LIN {X 0,Y 512.253,Z 580.66,A -85,B 0,C 180,E1 4907.429,E2 4907.429} C_VEL
LIN {X 0,Y 512.3,Z 580.66,A -85,B 0,C 180,E1 4912.681,E2 4912.681} C_VEL
LIN {X 0,Y 512.412,Z 580.694,A -85,B 0,C 180,E1 4919.232,E2 4919.232} C_VEL
LIN {X 0,Y 523.878,Z 610.794,A -85,B 0,C 180,E1 4920.286,E2 4920.286} C_VEL
LIN {X 0,Y 523.206,Z 668.635,A -85,B 0,C 180,E1 4921.275,E2 4921.275} C_VEL
LIN {X 0,Y 521.819,Z 705.735,A -85,B 0,C 180,E1 4922.556,E2 4922.556} C_VEL
LIN {X 0,Y 520.117,Z 737.921,A -85,B 0,C 180,E1 4924.318,E2 4924.318} C_VEL
LIN {X 0,Y 518.031,Z 770.325,A -85,B 0,C 180,E1 4926.817,E2 4926.817} C_VEL
LIN {X 0,Y 516.114,Z 799.539,A -85,B 0,C 180,E1 4929.907,E2 4929.907} C_VEL
LIN {X 0,Y 514.641,Z 823.98,A -85,B 0,C 180,E1 4933.388,E2 4933.388} C_VEL
LIN {X 0,Y 513.732,Z 843.903,A -85,B 0,C 180,E1 4937.273,E2 4937.273} C_VEL
LIN {X 0,Y 513.324,Z 857.536,A -85,B 0,C 180,E1 4941.121,E2 4941.121} C_VEL
LIN {X 0,Y 513.093,Z 865.986,A -85,B 0,C 180,E1 4944.937,E2 4944.937} C_VEL
LIN {X 0,Y 513.009,Z 869.513,A -85,B 0,C 180,E1 4948.313,E2 4948.313} C_VEL
LIN {X 0,Y 513.17,Z 869.515,A -85,B 0,C 180,E1 4951.684,E2 4951.684} C_VEL
LIN {X 0,Y 513.084,Z 864.493,A -85,B 0,C 180,E1 4955.907,E2 4955.907} C_VEL
LIN {X 0,Y 513.297,Z 854.958,A -85,B 0,C 180,E1 4959.725,E2 4959.725} C_VEL
LIN {X 0,Y 513.845,Z 840.043,A -85,B 0,C 180,E1 4963.586,E2 4963.586} C_VEL
LIN {X 0,Y 514.932,Z 818.765,A -85,B 0,C 180,E1 4967.453,E2 4967.453} C_VEL
LIN {X 0,Y 516.498,Z 792.754,A -85,B 0,C 180,E1 4970.897,E2 4970.897} C_VEL
LIN {X 0,Y 518.496,Z 762.754,A -85,B 0,C 180,E1 4973.845,E2 4973.845} C_VEL
LIN {X 0,Y 520.653,Z 728.929,A -85,B 0,C 180,E1 4976.245,E2 4976.245} C_VEL
LIN {X 0,Y 522.289,Z 696.341,A -85,B 0,C 180,E1 4977.831,E2 4977.831} C_VEL
LIN {X 0,Y 523.448,Z 660.966,A -85,B 0,C 180,E1 4978.906,E2 4978.906} C_VEL
LIN {X 0,Y 522.927,Z 606.604,A -85,B 0,C 180,E1 4979.824,E2 4979.824} C_VEL
LIN {X 0,Y 512.41,Z 580.66,A -85,B 0,C 180,E1 4980.856,E2 4980.856} C_VEL
LIN {X 0,Y 512.162,Z 580.66,A -85,B 0,C 180,E1 4987.298,E2 4987.298} C_VEL
LIN {X 0,Y 512.152,Z 580.66,A -85,B 0,C 180,E1 4992.657,E2 4992.657} C_VEL
LIN {X 0,Y 512.248,Z 580.66,A -85,B 0,C 180,E1 4997.425,E2 4997.425} C_VEL
LIN {X 0,Y 512.288,Z 580.66,A -85,B 0,C 180,E1 5002.678,E2 5002.678} C_VEL
LIN {X 0,Y 512.29,Z 580.66,A -85,B 0,C 180,E1 5008.666,E2 5008.666} C_VEL
LIN {X 0,Y 512.346,Z 580.66,A -85,B 0,C 180,E1 5013.781,E2 5013.781} C_VEL
LIN {X 0,Y 512.529,Z 580.66,A -85,B 0,C 180,E1 5019.309,E2 5019.309} C_VEL
LIN {X 0,Y 512.44,Z 580.66,A -85,B 0,C 180,E1 5024.63,E2 5024.63} C_VEL
LIN {X 0,Y 512.603,Z 580.66,A -85,B 0,C 180,E1 5029.824,E2 5029.824} C_VEL
LIN {X 0,Y 512.797,Z 580.66,A -85,B 0,C 180,E1 5034.933,E2 5034.933} C_VEL
LIN {X 0,Y 512.816,Z 580.66,A -85,B 0,C 180,E1 5039.997,E2 5039.997} C_VEL
LIN {X 0,Y 512.808,Z 580.66,A -85,B 0,C 180,E1 5045.061,E2 5045.061} C_VEL
LIN {X 0,Y 512.654,Z 580.66,A -85,B 0,C 180,E1 5050.168,E2 5050.168} C_VEL
LIN {X 0,Y 512.572,Z 580.66,A -85,B 0,C 180,E1 5055.36,E2 5055.36} C_VEL
LIN {X 0,Y 512.505,Z 580.66,A -85,B 0,C 180,E1 5060.685,E2 5060.685} C_VEL
LIN {X 0,Y 512.3,Z 580.66,A -85,B 0,C 180,E1 5066.215,E2 5066.215} C_VEL
LIN {X 0,Y 512.314,Z 580.66,A -85,B 0,C 180,E1 5072.011,E2 5072.011} C_VEL
LIN {X 0,Y 512.156,Z 580.66,A -85,B 0,C 180,E1 5078.216,E2 5078.216} C_VEL
LIN {X 0,Y 512.205,Z 580.66,A -85,B 0,C 180,E1 5085.009,E2 5085.009} C_VEL
LIN {X 0,Y 512.33,Z 580.66,A -85,B 0,C 180,E1 5089.967,E2 5089.967} C_VEL
LIN {X 0,Y 512.203,Z 580.66,A -85,B 0,C 180,E1 5095.965,E2 5095.965} C_VEL
LIN {X 0,Y 512.325,Z 580.66,A -85,B 0,C 180,E1 5102.065,E2 5102.065} C_VEL
LIN {X 0,Y 512.487,Z 581.105,A -85,B 0,C 180,E1 5106.168,E2 5106.168} C_VEL
LIN {X 0,Y 520.386,Z 606.411,A -85,B 0,C 180,E1 5107.997,E2 5107.997} C_VEL
LIN {X 0,Y 518.562,Z 636.165,A -85,B 0,C 180,E1 5110.12,E2 5110.12} C_VEL
LIN {X 0,Y 516.609,Z 662.595,A -85,B 0,C 180,E1 5112.838,E2 5112.838} C_VEL
LIN {X 0,Y 514.974,Z 684.992,A -85,B 0,C 180,E1 5116.076,E2 5116.076} C_VEL
LIN {X 0,Y 514.025,Z 701.113,A -85,B 0,C 180,E1 5119.369,E2 5119.369} C_VEL
LIN {X 0,Y 513.36,Z 713.574,A -85,B 0,C 180,E1 5123.249,E2 5123.249} C_VEL
LIN {X 0,Y 513.2,Z 719.653,A -85,B 0,C 180,E1 5126.63,E2 5126.63} C_VEL
LIN {X 0,Y 513.129,Z 721.603,A -85,B 0,C 180,E1 5130.001,E2 5130.001} C_VEL
LIN {X 0,Y 513.261,Z 718.398,A -85,B 0,C 180,E1 5134.216,E2 5134.216} C_VEL
LIN {X 0,Y 513.649,Z 709.866,A -85,B 0,C 180,E1 5138.023,E2 5138.023} C_VEL
LIN {X 0,Y 514.382,Z 695.343,A -85,B 0,C 180,E1 5141.851,E2 5141.851} C_VEL
LIN {X 0,Y 515.675,Z 676.023,A -85,B 0,C 180,E1 5145.27,E2 5145.27} C_VEL
LIN {X 0,Y 517.397,Z 652.213,A -85,B 0,C 180,E1 5148.252,E2 5148.252} C_VEL
LIN {X 0,Y 519.312,Z 624.854,A -85,B 0,C 180,E1 5150.69,E2 5150.69} C_VEL
LIN {X 0,Y 519.753,Z 602.818,A -85,B 0,C 180,E1 5152.175,E2 5152.175} C_VEL
LIN {X 0,Y 512.463,Z 580.66,A -85,B 0,C 180,E1 5153.799,E2 5153.799} C_VEL
LIN {X 0,Y 512.211,Z 580.66,A -85,B 0,C 180,E1 5160.055,E2 5160.055} C_VEL
LIN {X 0,Y 512.277,Z 580.66,A -85,B 0,C 180,E1 5166.095,E2 5166.095} C_VEL
LIN {X 0,Y 512.262,Z 580.66,A -85,B 0,C 180,E1 5170.395,E2 5170.395} C_VEL
LIN {X 0,Y 512.215,Z 580.66,A -85,B 0,C 180,E1 5177.354,E2 5177.354} C_VEL
LIN {X 0,Y 512.267,Z 580.66,A -85,B 0,C 180,E1 5182.686,E2 5182.686} C_VEL
LIN {X 0,Y 512.256,Z 580.66,A -85,B 0,C 180,E1 5188.678,E2 5188.678} C_VEL
LIN {X 0,Y 512.315,Z 580.66,A -85,B 0,C 180,E1 5193.786,E2 5193.786} C_VEL
LIN {X 0,Y 512.532,Z 580.66,A -85,B 0,C 180,E1 5199.316,E2 5199.316} C_VEL
LIN {X 0,Y 512.402,Z 580.66,A -85,B 0,C 180,E1 5204.635,E2 5204.635} C_VEL
LIN {X 0,Y 512.58,Z 580.66,A -85,B 0,C 180,E1 5209.83,E2 5209.83} C_VEL
LIN {X 0,Y 512.817,Z 580.66,A -85,B 0,C 180,E1 5214.939,E2 5214.939} C_VEL
LIN {X 0,Y 512.839,Z 580.66,A -85,B 0,C 180,E1 5220.003,E2 5220.003} C_VEL
LIN {X 0,Y 512.786,Z 580.66,A -85,B 0,C 180,E1 5225.068,E2 5225.068} C_VEL
LIN {X 0,Y 512.686,Z 580.66,A -85,B 0,C 180,E1 5230.174,E2 5230.174} C_VEL
LIN {X 0,Y 512.577,Z 580.66,A -85,B 0,C 180,E1 5235.366,E2 5235.366} C_VEL
LIN {X 0,Y 512.513,Z 580.66,A -85,B 0,C 180,E1 5240.692,E2 5240.692} C_VEL
LIN {X 0,Y 512.325,Z 580.66,A -85,B 0,C 180,E1 5246.22,E2 5246.22} C_VEL
LIN {X 0,Y 512.285,Z 580.66,A -85,B 0,C 180,E1 5252.02,E2 5252.02} C_VEL
LIN {X 0,Y 512.168,Z 580.66,A -85,B 0,C 180,E1 5258.088,E2 5258.088} C_VEL
LIN {X 0,Y 509.69,Z 580.66,A -85,B 0,C 180,E1 5259.518,E2 5259.518} C_VEL
LIN {X 0,Y 504.13,Z 580.66,A -85,B 0,C 180,E1 5261.908,E2 5261.908} C_VEL
LIN {X 0,Y 504.239,Z 580.66,A -85,B 0,C 180,E1 5266.505,E2 5266.505} C_VEL
LIN {X 0,Y 504.372,Z 580.66,A -85,B 0,C 180,E1 5271.077,E2 5271.077} C_VEL
LIN {X 0,Y 504.318,Z 580.66,A -85,B 0,C 180,E1 5276.907,E2 5276.907} C_VEL
LIN {X 0,Y 504.516,Z 580.66,A -85,B 0,C 180,E1 5278.767,E2 5278.767} C_VEL
LIN {X 0,Y 516.691,Z 611.482,A -85,B 0,C 180,E1 5279.931,E2 5279.931} C_VEL
LIN {X 0,Y 516.001,Z 667.111,A -85,B 0,C 180,E1 5280.899,E2 5280.899} C_VEL
LIN {X 0,Y 514.493,Z 704.279,A -85,B 0,C 180,E1 5282.191,E2 5282.191} C_VEL
LIN {X 0,Y 512.569,Z 740.82,A -85,B 0,C 180,E1 5284.163,E2 5284.163} C_VEL
LIN {X 0,Y 510.618,Z 770.896,A -85,B 0,C 180,E1 5286.513,E2 5286.513} C_VEL
LIN {X 0,Y 508.548,Z 799.538,A -85,B 0,C 180,E1 5289.595,E2 5289.595} C_VEL
LIN {X 0,Y 506.924,Z 823.979,A -85,B 0,C 180,E1 5293.127,E2 5293.127} C_VEL
LIN {X 0,Y 505.91,Z 843.903,A -85,B 0,C 180,E1 5297.072,E2 5297.072} C_VEL
LIN {X 0,Y 505.476,Z 856.878,A -85,B 0,C 180,E1 5300.746,E2 5300.746} C_VEL
LIN {X 0,Y 505.195,Z 865.986,A -85,B 0,C 180,E1 5304.858,E2 5304.858} C_VEL
LIN {X 0,Y 505.107,Z 869.513,A -85,B 0,C 180,E1 5308.287,E2 5308.287} C_VEL
LIN {X 0,Y 505.266,Z 869.515,A -85,B 0,C 180,E1 5311.71,E2 5311.71} C_VEL
LIN {X 0,Y 505.202,Z 864.492,A -85,B 0,C 180,E1 5315.999,E2 5315.999} C_VEL
LIN {X 0,Y 505.451,Z 854.946,A -85,B 0,C 180,E1 5319.882,E2 5319.882} C_VEL
LIN {X 0,Y 506.033,Z 840.042,A -85,B 0,C 180,E1 5323.799,E2 5323.799} C_VEL
LIN {X 0,Y 507.212,Z 819.028,A -85,B 0,C 180,E1 5327.686,E2 5327.686} C_VEL
LIN {X 0,Y 508.884,Z 793.85,A -85,B 0,C 180,E1 5331.094,E2 5331.094} C_VEL
LIN {X 0,Y 510.995,Z 764.887,A -85,B 0,C 180,E1 5334.021,E2 5334.021} C_VEL
LIN {X 0,Y 512.854,Z 735.228,A -85,B 0,C 180,E1 5336.187,E2 5336.187} C_VEL
LIN {X 0,Y 514.807,Z 698.308,A -85,B 0,C 180,E1 5338.068,E2 5338.068} C_VEL
LIN {X 0,Y 516.207,Z 660.797,A -85,B 0,C 180,E1 5339.253,E2 5339.253} C_VEL
LIN {X 0,Y 515.751,Z 608.845,A -85,B 0,C 180,E1 5340.157,E2 5340.157} C_VEL
LIN {X 0,Y 504.502,Z 580.66,A -85,B 0,C 180,E1 5341.293,E2 5341.293} C_VEL
LIN {X 0,Y 504.25,Z 580.66,A -85,B 0,C 180,E1 5346.759,E2 5346.759} C_VEL
LIN {X 0,Y 504.17,Z 580.66,A -85,B 0,C 180,E1 5353.498,E2 5353.498} C_VEL
LIN {X 0,Y 504.303,Z 580.66,A -85,B 0,C 180,E1 5358.83,E2 5358.83} C_VEL
LIN {X 0,Y 504.32,Z 580.66,A -85,B 0,C 180,E1 5365.354,E2 5365.354} C_VEL
LIN {X 0,Y 504.371,Z 580.66,A -85,B 0,C 180,E1 5371.399,E2 5371.399} C_VEL
LIN {X 0,Y 504.508,Z 580.66,A -85,B 0,C 180,E1 5377.994,E2 5377.994} C_VEL
LIN {X 0,Y 504.663,Z 580.66,A -85,B 0,C 180,E1 5383.089,E2 5383.089} C_VEL
LIN {X 0,Y 504.679,Z 580.66,A -85,B 0,C 180,E1 5389.663,E2 5389.663} C_VEL
LIN {X 0,Y 504.885,Z 580.66,A -85,B 0,C 180,E1 5394.853,E2 5394.853} C_VEL
LIN {X 0,Y 504.915,Z 580.66,A -85,B 0,C 180,E1 5399.997,E2 5399.997} C_VEL
LIN {X 0,Y 504.892,Z 580.66,A -85,B 0,C 180,E1 5405.141,E2 5405.141} C_VEL
LIN {X 0,Y 504.743,Z 580.66,A -85,B 0,C 180,E1 5410.329,E2 5410.329} C_VEL
LIN {X 0,Y 504.644,Z 580.66,A -85,B 0,C 180,E1 5415.607,E2 5415.607} C_VEL
LIN {X 0,Y 504.55,Z 580.66,A -85,B 0,C 180,E1 5421.027,E2 5421.027} C_VEL
LIN {X 0,Y 504.378,Z 580.66,A -85,B 0,C 180,E1 5426.659,E2 5426.659} C_VEL
LIN {X 0,Y 504.312,Z 580.66,A -85,B 0,C 180,E1 5433.098,E2 5433.098} C_VEL
LIN {X 0,Y 504.228,Z 580.66,A -85,B 0,C 180,E1 5438.929,E2 5438.929} C_VEL
LIN {X 0,Y 504.255,Z 580.66,A -85,B 0,C 180,E1 5445.897,E2 5445.897} C_VEL
LIN {X 0,Y 504.362,Z 580.66,A -85,B 0,C 180,E1 5451.08,E2 5451.08} C_VEL
LIN {X 0,Y 504.252,Z 580.66,A -85,B 0,C 180,E1 5456.906,E2 5456.906} C_VEL
LIN {X 0,Y 504.407,Z 580.66,A -85,B 0,C 180,E1 5463.34,E2 5463.34} C_VEL
LIN {X 0,Y 504.539,Z 581.013,A -85,B 0,C 180,E1 5465.648,E2 5465.648} C_VEL
LIN {X 0,Y 513.395,Z 608.606,A -85,B 0,C 180,E1 5467.666,E2 5467.666} C_VEL
LIN {X 0,Y 511.416,Z 638.199,A -85,B 0,C 180,E1 5469.83,E2 5469.83} C_VEL
LIN {X 0,Y 509.29,Z 664.127,A -85,B 0,C 180,E1 5472.552,E2 5472.552} C_VEL
LIN {X 0,Y 507.558,Z 685.323,A -85,B 0,C 180,E1 5475.657,E2 5475.657} C_VEL
LIN {X 0,Y 506.328,Z 702.896,A -85,B 0,C 180,E1 5479.311,E2 5479.311} C_VEL
LIN {X 0,Y 505.616,Z 714.835,A -85,B 0,C 180,E1 5483.146,E2 5483.146} C_VEL
LIN {X 0,Y 505.418,Z 720.857,A -85,B 0,C 180,E1 5486.578,E2 5486.578} C_VEL
LIN {X 0,Y 505.32,Z 722.79,A -85,B 0,C 180,E1 5490.001,E2 5490.001} C_VEL
LIN {X 0,Y 505.489,Z 719.611,A -85,B 0,C 180,E1 5494.281,E2 5494.281} C_VEL
LIN {X 0,Y 505.914,Z 711.171,A -85,B 0,C 180,E1 5498.146,E2 5498.146} C_VEL
LIN {X 0,Y 506.76,Z 696.769,A -85,B 0,C 180,E1 5502.032,E2 5502.032} C_VEL
LIN {X 0,Y 508.234,Z 677.656,A -85,B 0,C 180,E1 5505.499,E2 5505.499} C_VEL
LIN {X 0,Y 510.182,Z 653.532,A -85,B 0,C 180,E1 5508.583,E2 5508.583} C_VEL
LIN {X 0,Y 512.212,Z 627.084,A -85,B 0,C 180,E1 5510.99,E2 5510.99} C_VEL
LIN {X 0,Y 512.777,Z 605.367,A -85,B 0,C 180,E1 5512.493,E2 5512.493} C_VEL
LIN {X 0,Y 504.501,Z 580.66,A -85,B 0,C 180,E1 5514.355,E2 5514.355} C_VEL
LIN {X 0,Y 504.298,Z 580.66,A -85,B 0,C 180,E1 5520.576,E2 5520.576} C_VEL
LIN {X 0,Y 504.39,Z 580.66,A -85,B 0,C 180,E1 5526.751,E2 5526.751} C_VEL
LIN {X 0,Y 504.21,Z 580.66,A -85,B 0,C 180,E1 5531.576,E2 5531.576} C_VEL
LIN {X 0,Y 504.202,Z 580.66,A -85,B 0,C 180,E1 5536.509,E2 5536.509} C_VEL
LIN {X 0,Y 504.338,Z 580.66,A -85,B 0,C 180,E1 5541.081,E2 5541.081} C_VEL
LIN {X 0,Y 504.248,Z 580.66,A -85,B 0,C 180,E1 5546.919,E2 5546.919} C_VEL
LIN {X 0,Y 504.386,Z 580.66,A -85,B 0,C 180,E1 5553.342,E2 5553.342} C_VEL
LIN {X 0,Y 504.57,Z 580.66,A -85,B 0,C 180,E1 5558.974,E2 5558.974} C_VEL
LIN {X 0,Y 504.499,Z 580.66,A -85,B 0,C 180,E1 5564.388,E2 5564.388} C_VEL
LIN {X 0,Y 504.65,Z 580.66,A -85,B 0,C 180,E1 5570.657,E2 5570.657} C_VEL
LIN {X 0,Y 504.846,Z 580.66,A -85,B 0,C 180,E1 5576.576,E2 5576.576} C_VEL
LIN {X 0,Y 504.793,Z 580.66,A -85,B 0,C 180,E1 5581.716,E2 5581.716} C_VEL
LIN {X 0,Y 504.771,Z 580.66,A -85,B 0,C 180,E1 5586.87,E2 5586.87} C_VEL
LIN {X 0,Y 504.713,Z 580.66,A -85,B 0,C 180,E1 5592.083,E2 5592.083} C_VEL
LIN {X 0,Y 504.628,Z 580.66,A -85,B 0,C 180,E1 5597.401,E2 5597.401} C_VEL
LIN {X 0,Y 504.49,Z 580.66,A -85,B 0,C 180,E1 5602.884,E2 5602.884} C_VEL
LIN {X 0,Y 504.366,Z 580.66,A -85,B 0,C 180,E1 5608.601,E2 5608.601} C_VEL
LIN {X 0,Y 504.309,Z 580.66,A -85,B 0,C 180,E1 5614.647,E2 5614.647} C_VEL
LIN {X 0,Y 504.177,Z 580.66,A -85,B 0,C 180,E1 5621.182,E2 5621.182} C_VEL
LIN {X 0,Y 504.13,Z 580.66,A -85,B 0,C 180,E1 5621.908,E2 5621.908} C_VEL
LIN {X 0,Y 500.222,Z 580.66,A -85,B 0,C 180,E1 5623.857,E2 5623.857} C_VEL
LIN {X 0,Y 496.32,Z 580.66,A -85,B 0,C 180,E1 5625.837,E2 5625.837} C_VEL
LIN {X 0,Y 496.42,Z 580.66,A -85,B 0,C 180,E1 5632.216,E2 5632.216} C_VEL
LIN {X 0,Y 496.608,Z 581.359,A -85,B 0,C 180,E1 5638.366,E2 5638.366} C_VEL
LIN {X 0,Y 509.556,Z 615.391,A -85,B 0,C 180,E1 5639.618,E2 5639.618} C_VEL
LIN {X 0,Y 508.758,Z 666.961,A -85,B 0,C 180,E1 5640.55,E2 5640.55} C_VEL
LIN {X 0,Y 507.091,Z 704.06,A -85,B 0,C 180,E1 5641.87,E2 5641.87} C_VEL
LIN {X 0,Y 505.01,Z 740.835,A -85,B 0,C 180,E1 5643.9,E2 5643.9} C_VEL
LIN {X 0,Y 502.786,Z 774.814,A -85,B 0,C 180,E1 5646.58,E2 5646.58} C_VEL
LIN {X 0,Y 500.904,Z 800.388,A -85,B 0,C 180,E1 5649.381,E2 5649.381} C_VEL
LIN {X 0,Y 499.198,Z 823.978,A -85,B 0,C 180,E1 5652.858,E2 5652.858} C_VEL
LIN {X 0,Y 498.11,Z 843.903,A -85,B 0,C 180,E1 5656.866,E2 5656.866} C_VEL
LIN {X 0,Y 497.509,Z 858.68,A -85,B 0,C 180,E1 5661.276,E2 5661.276} C_VEL
LIN {X 0,Y 497.286,Z 867.19,A -85,B 0,C 180,E1 5665.648,E2 5665.648} C_VEL
LIN {X 0,Y 497.23,Z 870,A -85,B 0,C 180,E1 5669.999,E2 5669.999} C_VEL
LIN {X 0,Y 497.302,Z 867.196,A -85,B 0,C 180,E1 5674.349,E2 5674.349} C_VEL
LIN {X 0,Y 497.476,Z 858.684,A -85,B 0,C 180,E1 5678.721,E2 5678.721} C_VEL
LIN {X 0,Y 497.926,Z 845.658,A -85,B 0,C 180,E1 5682.69,E2 5682.69} C_VEL
LIN {X 0,Y 498.973,Z 826.619,A -85,B 0,C 180,E1 5686.694,E2 5686.694} C_VEL
LIN {X 0,Y 500.71,Z 802.092,A -85,B 0,C 180,E1 5690.402,E2 5690.402} C_VEL
LIN {X 0,Y 502.633,Z 777.24,A -85,B 0,C 180,E1 5693.194,E2 5693.194} C_VEL
LIN {X 0,Y 504.826,Z 744.141,A -85,B 0,C 180,E1 5695.869,E2 5695.869} C_VEL
LIN {X 0,Y 506.887,Z 707.945,A -85,B 0,C 180,E1 5697.958,E2 5697.958} C_VEL
LIN {X 0,Y 508.596,Z 670.167,A -85,B 0,C 180,E1 5699.364,E2 5699.364} C_VEL
LIN {X 0,Y 509.328,Z 625.381,A -85,B 0,C 180,E1 5700.239,E2 5700.239} C_VEL
LIN {X 0,Y 508.58,Z 611.103,A -85,B 0,C 180,E1 5700.501,E2 5700.501} C_VEL
LIN {X 0,Y 496.558,Z 580.66,A -85,B 0,C 180,E1 5701.693,E2 5701.693} C_VEL
LIN {X 0,Y 496.248,Z 580.66,A -85,B 0,C 180,E1 5707.759,E2 5707.759} C_VEL
LIN {X 0,Y 496.301,Z 580.66,A -85,B 0,C 180,E1 5714.367,E2 5714.367} C_VEL
LIN {X 0,Y 496.38,Z 580.66,A -85,B 0,C 180,E1 5720.327,E2 5720.327} C_VEL
LIN {X 0,Y 496.377,Z 580.66,A -85,B 0,C 180,E1 5726.824,E2 5726.824} C_VEL
LIN {X 0,Y 496.458,Z 580.66,A -85,B 0,C 180,E1 5732.874,E2 5732.874} C_VEL
LIN {X 0,Y 496.637,Z 580.66,A -85,B 0,C 180,E1 5738.615,E2 5738.615} C_VEL
LIN {X 0,Y 496.647,Z 580.66,A -85,B 0,C 180,E1 5744.128,E2 5744.128} C_VEL
LIN {X 0,Y 496.75,Z 580.66,A -85,B 0,C 180,E1 5749.496,E2 5749.496} C_VEL
LIN {X 0,Y 496.987,Z 580.66,A -85,B 0,C 180,E1 5754.771,E2 5754.771} C_VEL
LIN {X 0,Y 497.022,Z 580.66,A -85,B 0,C 180,E1 5759.997,E2 5759.997} C_VEL
LIN {X 0,Y 496.987,Z 580.66,A -85,B 0,C 180,E1 5765.222,E2 5765.222} C_VEL
LIN {X 0,Y 496.817,Z 580.66,A -85,B 0,C 180,E1 5770.496,E2 5770.496} C_VEL
LIN {X 0,Y 496.733,Z 580.66,A -85,B 0,C 180,E1 5775.862,E2 5775.862} C_VEL
LIN {X 0,Y 496.621,Z 580.66,A -85,B 0,C 180,E1 5781.379,E2 5781.379} C_VEL
LIN {X 0,Y 496.418,Z 580.66,A -85,B 0,C 180,E1 5787.121,E2 5787.121} C_VEL
LIN {X 0,Y 496.405,Z 580.66,A -85,B 0,C 180,E1 5793.166,E2 5793.166} C_VEL
LIN {X 0,Y 496.222,Z 580.66,A -85,B 0,C 180,E1 5799.679,E2 5799.679} C_VEL
LIN {X 0,Y 496.334,Z 580.66,A -85,B 0,C 180,E1 5805.637,E2 5805.637} C_VEL
LIN {X 0,Y 496.403,Z 580.66,A -85,B 0,C 180,E1 5812.208,E2 5812.208} C_VEL
LIN {X 0,Y 496.316,Z 580.66,A -85,B 0,C 180,E1 5818.34,E2 5818.34} C_VEL
LIN {X 0,Y 496.522,Z 580.66,A -85,B 0,C 180,E1 5824.822,E2 5824.822} C_VEL
LIN {X 0,Y 496.596,Z 581.594,A -85,B 0,C 180,E1 5825.148,E2 5825.148} C_VEL
LIN {X 0,Y 506.22,Z 610.107,A -85,B 0,C 180,E1 5827.287,E2 5827.287} C_VEL
LIN {X 0,Y 504.243,Z 640.16,A -85,B 0,C 180,E1 5829.53,E2 5829.53} C_VEL
LIN {X 0,Y 501.927,Z 666.279,A -85,B 0,C 180,E1 5832.334,E2 5832.334} C_VEL
LIN {X 0,Y 500.02,Z 687.497,A -85,B 0,C 180,E1 5835.55,E2 5835.55} C_VEL
LIN {X 0,Y 498.684,Z 704.107,A -85,B 0,C 180,E1 5839.101,E2 5839.101} C_VEL
LIN {X 0,Y 497.871,Z 716.1,A -85,B 0,C 180,E1 5843.038,E2 5843.038} C_VEL
LIN {X 0,Y 497.63,Z 722.064,A -85,B 0,C 180,E1 5846.525,E2 5846.525} C_VEL
LIN {X 0,Y 497.532,Z 723.973,A -85,B 0,C 180,E1 5850.001,E2 5850.001} C_VEL
LIN {X 0,Y 497.714,Z 720.826,A -85,B 0,C 180,E1 5854.348,E2 5854.348} C_VEL
LIN {X 0,Y 498.182,Z 712.466,A -85,B 0,C 180,E1 5858.273,E2 5858.273} C_VEL
LIN {X 0,Y 499.167,Z 698.228,A -85,B 0,C 180,E1 5862.218,E2 5862.218} C_VEL
LIN {X 0,Y 500.797,Z 679.309,A -85,B 0,C 180,E1 5865.736,E2 5865.736} C_VEL
LIN {X 0,Y 502.922,Z 655.399,A -85,B 0,C 180,E1 5868.862,E2 5868.862} C_VEL
LIN {X 0,Y 505.197,Z 627.918,A -85,B 0,C 180,E1 5871.394,E2 5871.394} C_VEL
LIN {X 0,Y 505.961,Z 608.702,A -85,B 0,C 180,E1 5872.729,E2 5872.729} C_VEL
LIN {X 0,Y 496.531,Z 580.66,A -85,B 0,C 180,E1 5874.825,E2 5874.825} C_VEL
LIN {X 0,Y 496.325,Z 580.66,A -85,B 0,C 180,E1 5881.122,E2 5881.122} C_VEL
LIN {X 0,Y 496.4,Z 580.66,A -85,B 0,C 180,E1 5887.443,E2 5887.443} C_VEL
LIN {X 0,Y 496.249,Z 580.66,A -85,B 0,C 180,E1 5893.141,E2 5893.141} C_VEL
LIN {X 0,Y 496.319,Z 580.66,A -85,B 0,C 180,E1 5899.471,E2 5899.471} C_VEL
LIN {X 0,Y 496.378,Z 580.66,A -85,B 0,C 180,E1 5905.163,E2 5905.163} C_VEL
LIN {X 0,Y 496.384,Z 580.66,A -85,B 0,C 180,E1 5911.833,E2 5911.833} C_VEL
LIN {X 0,Y 496.513,Z 580.66,A -85,B 0,C 180,E1 5916.734,E2 5916.734} C_VEL
LIN {X 0,Y 496.728,Z 580.66,A -85,B 0,C 180,E1 5922.32,E2 5922.32} C_VEL
LIN {X 0,Y 496.729,Z 580.66,A -85,B 0,C 180,E1 5929.502,E2 5929.502} C_VEL
LIN {X 0,Y 497.007,Z 580.66,A -85,B 0,C 180,E1 5934.778,E2 5934.778} C_VEL
LIN {X 0,Y 497.044,Z 580.66,A -85,B 0,C 180,E1 5940.003,E2 5940.003} C_VEL
LIN {X 0,Y 496.972,Z 580.66,A -85,B 0,C 180,E1 5945.229,E2 5945.229} C_VEL
LIN {X 0,Y 496.85,Z 580.66,A -85,B 0,C 180,E1 5950.502,E2 5950.502} C_VEL
LIN {X 0,Y 496.725,Z 580.66,A -85,B 0,C 180,E1 5955.869,E2 5955.869} C_VEL
LIN {X 0,Y 496.636,Z 580.66,A -85,B 0,C 180,E1 5961.385,E2 5961.385} C_VEL
LIN {X 0,Y 496.45,Z 580.66,A -85,B 0,C 180,E1 5967.126,E2 5967.126} C_VEL
LIN {X 0,Y 496.388,Z 580.66,A -85,B 0,C 180,E1 5973.175,E2 5973.175} C_VEL
LIN {X 0,Y 496.23,Z 580.66,A -85,B 0,C 180,E1 5979.687,E2 5979.687} C_VEL
LIN {X 0,Y 496.32,Z 580.66,A -85,B 0,C 180,E1 5985.837,E2 5985.837} C_VEL
LIN {X 0,Y 492.364,Z 580.66,A -85,B 0,C 180,E1 5987.811,E2 5987.811} C_VEL
LIN {X 0,Y 488.442,Z 580.66,A -85,B 0,C 180,E1 5989.816,E2 5989.816} C_VEL
LIN {X 0,Y 488.477,Z 580.66,A -85,B 0,C 180,E1 5996.217,E2 5996.217} C_VEL
LIN {X 0,Y 488.598,Z 581.283,A -85,B 0,C 180,E1 5997.887,E2 5997.887} C_VEL
LIN {X 0,Y 502.356,Z 615.662,A -85,B 0,C 180,E1 5999.241,E2 5999.241} C_VEL
LIN {X 0,Y 501.523,Z 666.523,A -85,B 0,C 180,E1 6000.185,E2 6000.185} C_VEL
LIN {X 0,Y 499.741,Z 702.563,A -85,B 0,C 180,E1 6001.48,E2 6001.48} C_VEL
LIN {X 0,Y 497.538,Z 739.366,A -85,B 0,C 180,E1 6003.532,E2 6003.532} C_VEL
LIN {X 0,Y 495.241,Z 772.505,A -85,B 0,C 180,E1 6006.162,E2 6006.162} C_VEL
LIN {X 0,Y 493.21,Z 800.895,A -85,B 0,C 180,E1 6009.188,E2 6009.188} C_VEL
LIN {X 0,Y 491.656,Z 821.333,A -85,B 0,C 180,E1 6012.126,E2 6012.126} C_VEL
LIN {X 0,Y 490.443,Z 840.028,A -85,B 0,C 180,E1 6015.75,E2 6015.75} C_VEL
LIN {X 0,Y 489.744,Z 855.451,A -85,B 0,C 180,E1 6019.967,E2 6019.967} C_VEL
LIN {X 0,Y 489.497,Z 864.486,A -85,B 0,C 180,E1 6023.805,E2 6023.805} C_VEL
LIN {X 0,Y 489.325,Z 869.512,A -85,B 0,C 180,E1 6028.231,E2 6028.231} C_VEL
LIN {X 0,Y 489.474,Z 869.514,A -85,B 0,C 180,E1 6031.765,E2 6031.765} C_VEL
LIN {X 0,Y 489.447,Z 864.492,A -85,B 0,C 180,E1 6036.193,E2 6036.193} C_VEL
LIN {X 0,Y 489.697,Z 855.533,A -85,B 0,C 180,E1 6040.005,E2 6040.005} C_VEL
LIN {X 0,Y 490.467,Z 840.041,A -85,B 0,C 180,E1 6044.246,E2 6044.246} C_VEL
LIN {X 0,Y 491.899,Z 819.149,A -85,B 0,C 180,E1 6048.236,E2 6048.236} C_VEL
LIN {X 0,Y 493.488,Z 796.447,A -85,B 0,C 180,E1 6051.355,E2 6051.355} C_VEL
LIN {X 0,Y 495.696,Z 765.715,A -85,B 0,C 180,E1 6054.444,E2 6054.444} C_VEL
LIN {X 0,Y 497.951,Z 732.522,A -85,B 0,C 180,E1 6056.907,E2 6056.907} C_VEL
LIN {X 0,Y 500.161,Z 696.283,A -85,B 0,C 180,E1 6058.798,E2 6058.798} C_VEL
LIN {X 0,Y 501.796,Z 658.508,A -85,B 0,C 180,E1 6060.018,E2 6060.018} C_VEL
LIN {X 0,Y 501.448,Z 613.288,A -85,B 0,C 180,E1 6060.857,E2 6060.857} C_VEL
LIN {X 0,Y 488.586,Z 580.66,A -85,B 0,C 180,E1 6062.218,E2 6062.218} C_VEL
LIN {X 0,Y 488.323,Z 580.66,A -85,B 0,C 180,E1 6068.168,E2 6068.168} C_VEL
LIN {X 0,Y 488.392,Z 580.66,A -85,B 0,C 180,E1 6074.714,E2 6074.714} C_VEL
LIN {X 0,Y 488.455,Z 580.66,A -85,B 0,C 180,E1 6080.558,E2 6080.558} C_VEL
LIN {X 0,Y 488.464,Z 580.66,A -85,B 0,C 180,E1 6086.515,E2 6086.515} C_VEL
LIN {X 0,Y 488.532,Z 580.66,A -85,B 0,C 180,E1 6092.397,E2 6092.397} C_VEL
LIN {X 0,Y 488.67,Z 580.66,A -85,B 0,C 180,E1 6098.249,E2 6098.249} C_VEL
LIN {X 0,Y 488.73,Z 580.66,A -85,B 0,C 180,E1 6103.864,E2 6103.864} C_VEL
LIN {X 0,Y 488.828,Z 580.66,A -85,B 0,C 180,E1 6109.324,E2 6109.324} C_VEL
LIN {X 0,Y 489.074,Z 580.66,A -85,B 0,C 180,E1 6114.686,E2 6114.686} C_VEL
LIN {X 0,Y 489.122,Z 580.66,A -85,B 0,C 180,E1 6119.997,E2 6119.997} C_VEL
LIN {X 0,Y 489.071,Z 580.66,A -85,B 0,C 180,E1 6125.307,E2 6125.307} C_VEL
LIN {X 0,Y 488.891,Z 580.66,A -85,B 0,C 180,E1 6130.668,E2 6130.668} C_VEL
LIN {X 0,Y 488.761,Z 580.66,A -85,B 0,C 180,E1 6136.861,E2 6136.861} C_VEL
LIN {X 0,Y 488.65,Z 580.66,A -85,B 0,C 180,E1 6142.127,E2 6142.127} C_VEL
LIN {X 0,Y 488.497,Z 580.66,A -85,B 0,C 180,E1 6147.598,E2 6147.598} C_VEL
LIN {X 0,Y 488.454,Z 580.66,A -85,B 0,C 180,E1 6153.778,E2 6153.778} C_VEL
LIN {X 0,Y 488.317,Z 580.66,A -85,B 0,C 180,E1 6160.453,E2 6160.453} C_VEL
LIN {X 0,Y 488.418,Z 580.66,A -85,B 0,C 180,E1 6167.185,E2 6167.185} C_VEL
LIN {X 0,Y 488.436,Z 580.66,A -85,B 0,C 180,E1 6173.43,E2 6173.43} C_VEL
LIN {X 0,Y 488.409,Z 580.66,A -85,B 0,C 180,E1 6179.878,E2 6179.878} C_VEL
LIN {X 0,Y 488.616,Z 581.156,A -85,B 0,C 180,E1 6184.59,E2 6184.59} C_VEL
LIN {X 0,Y 499.064,Z 611.96,A -85,B 0,C 180,E1 6186.938,E2 6186.938} C_VEL
LIN {X 0,Y 497.031,Z 641.874,A -85,B 0,C 180,E1 6189.219,E2 6189.219} C_VEL
LIN {X 0,Y 494.631,Z 667.725,A -85,B 0,C 180,E1 6192.034,E2 6192.034} C_VEL
LIN {X 0,Y 492.518,Z 689.061,A -85,B 0,C 180,E1 6195.325,E2 6195.325} C_VEL
LIN {X 0,Y 491.036,Z 705.495,A -85,B 0,C 180,E1 6198.929,E2 6198.929} C_VEL
LIN {X 0,Y 490.132,Z 717.374,A -85,B 0,C 180,E1 6202.928,E2 6202.928} C_VEL
LIN {X 0,Y 489.849,Z 723.27,A -85,B 0,C 180,E1 6206.469,E2 6206.469} C_VEL
LIN {X 0,Y 489.723,Z 725.16,A -85,B 0,C 180,E1 6210.001,E2 6210.001} C_VEL
LIN {X 0,Y 489.933,Z 722.044,A -85,B 0,C 180,E1 6214.417,E2 6214.417} C_VEL
LIN {X 0,Y 490.459,Z 713.789,A -85,B 0,C 180,E1 6218.405,E2 6218.405} C_VEL
LIN {X 0,Y 491.579,Z 699.686,A -85,B 0,C 180,E1 6222.409,E2 6222.409} C_VEL
LIN {X 0,Y 493.349,Z 680.929,A -85,B 0,C 180,E1 6225.979,E2 6225.979} C_VEL
LIN {X 0,Y 495.56,Z 657.962,A -85,B 0,C 180,E1 6229.05,E2 6229.05} C_VEL
LIN {X 0,Y 497.943,Z 630.97,A -85,B 0,C 180,E1 6231.622,E2 6231.622} C_VEL
LIN {X 0,Y 498.684,Z 610.457,A -85,B 0,C 180,E1 6233.093,E2 6233.093} C_VEL
LIN {X 0,Y 488.61,Z 580.66,A -85,B 0,C 180,E1 6235.34,E2 6235.34} C_VEL
LIN {X 0,Y 488.397,Z 580.66,A -85,B 0,C 180,E1 6241.685,E2 6241.685} C_VEL
LIN {X 0,Y 488.476,Z 580.66,A -85,B 0,C 180,E1 6248.158,E2 6248.158} C_VEL
LIN {X 0,Y 488.372,Z 580.66,A -85,B 0,C 180,E1 6254.721,E2 6254.721} C_VEL
LIN {X 0,Y 488.434,Z 580.66,A -85,B 0,C 180,E1 6260.565,E2 6260.565} C_VEL
LIN {X 0,Y 488.417,Z 580.66,A -85,B 0,C 180,E1 6266.529,E2 6266.529} C_VEL
LIN {X 0,Y 488.48,Z 580.66,A -85,B 0,C 180,E1 6272.401,E2 6272.401} C_VEL
LIN {X 0,Y 488.67,Z 580.66,A -85,B 0,C 180,E1 6278.256,E2 6278.256} C_VEL
LIN {X 0,Y 488.706,Z 580.66,A -85,B 0,C 180,E1 6283.87,E2 6283.87} C_VEL
LIN {X 0,Y 488.808,Z 580.66,A -85,B 0,C 180,E1 6289.33,E2 6289.33} C_VEL
LIN {X 0,Y 489.093,Z 580.66,A -85,B 0,C 180,E1 6294.693,E2 6294.693} C_VEL
LIN {X 0,Y 489.143,Z 580.66,A -85,B 0,C 180,E1 6300.003,E2 6300.003} C_VEL
LIN {X 0,Y 489.056,Z 580.66,A -85,B 0,C 180,E1 6305.314,E2 6305.314} C_VEL
LIN {X 0,Y 488.924,Z 580.66,A -85,B 0,C 180,E1 6310.674,E2 6310.674} C_VEL
LIN {X 0,Y 488.745,Z 580.66,A -85,B 0,C 180,E1 6316.844,E2 6316.844} C_VEL
LIN {X 0,Y 488.659,Z 580.66,A -85,B 0,C 180,E1 6322.122,E2 6322.122} C_VEL
LIN {X 0,Y 488.526,Z 580.66,A -85,B 0,C 180,E1 6327.603,E2 6327.603} C_VEL
LIN {X 0,Y 488.458,Z 580.66,A -85,B 0,C 180,E1 6333.785,E2 6333.785} C_VEL
LIN {X 0,Y 488.332,Z 580.66,A -85,B 0,C 180,E1 6340.46,E2 6340.46} C_VEL
LIN {X 0,Y 488.36,Z 580.66,A -85,B 0,C 180,E1 6345.831,E2 6345.831} C_VEL
LIN {X 0,Y 488.442,Z 580.66,A -85,B 0,C 180,E1 6349.816,E2 6349.816} C_VEL
LIN {X 0,Y 485.942,Z 580.66,A -85,B 0,C 180,E1 6351.328,E2 6351.328} C_VEL
LIN {X 0,Y 480.518,Z 580.66,A -85,B 0,C 180,E1 6353.859,E2 6353.859} C_VEL
LIN {X 0,Y 480.662,Z 581.316,A -85,B 0,C 180,E1 6357.39,E2 6357.39} C_VEL
LIN {X 0,Y 495.167,Z 617.768,A -85,B 0,C 180,E1 6358.884,E2 6358.884} C_VEL
LIN {X 0,Y 494.292,Z 665.78,A -85,B 0,C 180,E1 6359.807,E2 6359.807} C_VEL
LIN {X 0,Y 492.421,Z 701.316,A -85,B 0,C 180,E1 6361.102,E2 6361.102} C_VEL
LIN {X 0,Y 490.059,Z 738.353,A -85,B 0,C 180,E1 6363.184,E2 6363.184} C_VEL
LIN {X 0,Y 487.525,Z 772.575,A -85,B 0,C 180,E1 6365.957,E2 6365.957} C_VEL
LIN {X 0,Y 485.273,Z 802.452,A -85,B 0,C 180,E1 6369.248,E2 6369.248} C_VEL
LIN {X 0,Y 483.489,Z 827.744,A -85,B 0,C 180,E1 6373.023,E2 6373.023} C_VEL
LIN {X 0,Y 482.431,Z 844.396,A -85,B 0,C 180,E1 6376.56,E2 6376.56} C_VEL
LIN {X 0,Y 481.769,Z 858.68,A -85,B 0,C 180,E1 6380.989,E2 6380.989} C_VEL
LIN {X 0,Y 481.517,Z 867.189,A -85,B 0,C 180,E1 6385.505,E2 6385.505} C_VEL
LIN {X 0,Y 481.437,Z 870,A -85,B 0,C 180,E1 6389.998,E2 6389.998} C_VEL
LIN {X 0,Y 481.524,Z 867.195,A -85,B 0,C 180,E1 6394.492,E2 6394.492} C_VEL
LIN {X 0,Y 481.726,Z 858.684,A -85,B 0,C 180,E1 6399.009,E2 6399.009} C_VEL
LIN {X 0,Y 482.34,Z 844.375,A -85,B 0,C 180,E1 6403.448,E2 6403.448} C_VEL
LIN {X 0,Y 483.51,Z 826.502,A -85,B 0,C 180,E1 6407.202,E2 6407.202} C_VEL
LIN {X 0,Y 485.284,Z 801.367,A -85,B 0,C 180,E1 6410.887,E2 6410.887} C_VEL
LIN {X 0,Y 487.529,Z 772.563,A -85,B 0,C 180,E1 6414.043,E2 6414.043} C_VEL
LIN {X 0,Y 489.946,Z 739.612,A -85,B 0,C 180,E1 6416.728,E2 6416.728} C_VEL
LIN {X 0,Y 492.38,Z 702.522,A -85,B 0,C 180,E1 6418.843,E2 6418.843} C_VEL
LIN {X 0,Y 494.315,Z 665.33,A -85,B 0,C 180,E1 6420.207,E2 6420.207} C_VEL
LIN {X 0,Y 494.475,Z 616.025,A -85,B 0,C 180,E1 6421.195,E2 6421.195} C_VEL
LIN {X 0,Y 480.642,Z 580.66,A -85,B 0,C 180,E1 6422.652,E2 6422.652} C_VEL
LIN {X 0,Y 480.395,Z 580.66,A -85,B 0,C 180,E1 6428.915,E2 6428.915} C_VEL
LIN {X 0,Y 480.402,Z 580.66,A -85,B 0,C 180,E1 6433.743,E2 6433.743} C_VEL
LIN {X 0,Y 480.505,Z 580.66,A -85,B 0,C 180,E1 6438.906,E2 6438.906} C_VEL
LIN {X 0,Y 480.491,Z 580.66,A -85,B 0,C 180,E1 6444.733,E2 6444.733} C_VEL
LIN {X 0,Y 480.542,Z 580.66,A -85,B 0,C 180,E1 6449.838,E2 6449.838} C_VEL
LIN {X 0,Y 480.652,Z 580.66,A -85,B 0,C 180,E1 6455.911,E2 6455.911} C_VEL
LIN {X 0,Y 480.867,Z 580.66,A -85,B 0,C 180,E1 6461.709,E2 6461.709} C_VEL
LIN {X 0,Y 480.799,Z 580.66,A -85,B 0,C 180,E1 6467.307,E2 6467.307} C_VEL
LIN {X 0,Y 481.107,Z 580.66,A -85,B 0,C 180,E1 6472.79,E2 6472.79} C_VEL
LIN {X 0,Y 481.379,Z 580.66,A -85,B 0,C 180,E1 6478.2,E2 6478.2} C_VEL
LIN {X 0,Y 481.324,Z 580.66,A -85,B 0,C 180,E1 6483.591,E2 6483.591} C_VEL
LIN {X 0,Y 481.05,Z 580.66,A -85,B 0,C 180,E1 6489.02,E2 6489.02} C_VEL
LIN {X 0,Y 480.94,Z 580.66,A -85,B 0,C 180,E1 6494.532,E2 6494.532} C_VEL
LIN {X 0,Y 480.797,Z 580.66,A -85,B 0,C 180,E1 6500.191,E2 6500.191} C_VEL
LIN {X 0,Y 480.617,Z 580.66,A -85,B 0,C 180,E1 6506.069,E2 6506.069} C_VEL
LIN {X 0,Y 480.557,Z 580.66,A -85,B 0,C 180,E1 6512.256,E2 6512.256} C_VEL
LIN {X 0,Y 480.389,Z 580.66,A -85,B 0,C 180,E1 6518.912,E2 6518.912} C_VEL
LIN {X 0,Y 480.391,Z 580.66,A -85,B 0,C 180,E1 6523.746,E2 6523.746} C_VEL
LIN {X 0,Y 480.497,Z 580.66,A -85,B 0,C 180,E1 6528.902,E2 6528.902} C_VEL
LIN {X 0,Y 480.481,Z 580.66,A -85,B 0,C 180,E1 6534.728,E2 6534.728} C_VEL
LIN {X 0,Y 480.509,Z 580.66,A -85,B 0,C 180,E1 6539.84,E2 6539.84} C_VEL
LIN {X 0,Y 480.626,Z 580.946,A -85,B 0,C 180,E1 6544.03,E2 6544.03} C_VEL
LIN {X 0,Y 490.831,Z 610.731,A -85,B 0,C 180,E1 6546.307,E2 6546.307} C_VEL
LIN {X 0,Y 491.878,Z 619.119,A -85,B 0,C 180,E1 6546.956,E2 6546.956} C_VEL
LIN {X 0,Y 489.512,Z 647.05,A -85,B 0,C 180,E1 6549.24,E2 6549.24} C_VEL
LIN {X 0,Y 486.92,Z 672.355,A -85,B 0,C 180,E1 6552.182,E2 6552.182} C_VEL
LIN {X 0,Y 484.742,Z 693.115,A -85,B 0,C 180,E1 6555.582,E2 6555.582} C_VEL
LIN {X 0,Y 483.114,Z 709.503,A -85,B 0,C 180,E1 6559.497,E2 6559.497} C_VEL
LIN {X 0,Y 482.265,Z 720.468,A -85,B 0,C 180,E1 6563.715,E2 6563.715} C_VEL
LIN {X 0,Y 482.071,Z 724.477,A -85,B 0,C 180,E1 6566.412,E2 6566.412} C_VEL
LIN {X 0,Y 481.916,Z 726.346,A -85,B 0,C 180,E1 6570.002,E2 6570.002} C_VEL
LIN {X 0,Y 482.17,Z 723.262,A -85,B 0,C 180,E1 6574.489,E2 6574.489} C_VEL
LIN {X 0,Y 482.737,Z 715.098,A -85,B 0,C 180,E1 6578.54,E2 6578.54} C_VEL
LIN {X 0,Y 483.998,Z 701.118,A -85,B 0,C 180,E1 6582.607,E2 6582.607} C_VEL
LIN {X 0,Y 485.884,Z 682.395,A -85,B 0,C 180,E1 6586.232,E2 6586.232} C_VEL
LIN {X 0,Y 488.261,Z 659.502,A -85,B 0,C 180,E1 6589.346,E2 6589.346} C_VEL
LIN {X 0,Y 490.761,Z 633.006,A -85,B 0,C 180,E1 6591.926,E2 6591.926} C_VEL
LIN {X 0,Y 491.442,Z 612.514,A -85,B 0,C 180,E1 6593.44,E2 6593.44} C_VEL
LIN {X 0,Y 480.75,Z 581.988,A -85,B 0,C 180,E1 6595.828,E2 6595.828} C_VEL
LIN {X 0,Y 480.617,Z 580.66,A -85,B 0,C 180,E1 6596.076,E2 6596.076} C_VEL
LIN {X 0,Y 480.473,Z 580.66,A -85,B 0,C 180,E1 6602.27,E2 6602.27} C_VEL
LIN {X 0,Y 480.54,Z 580.66,A -85,B 0,C 180,E1 6608.905,E2 6608.905} C_VEL
LIN {X 0,Y 480.407,Z 580.66,A -85,B 0,C 180,E1 6613.753,E2 6613.753} C_VEL
LIN {X 0,Y 480.46,Z 580.66,A -85,B 0,C 180,E1 6618.917,E2 6618.917} C_VEL
LIN {X 0,Y 480.465,Z 580.66,A -85,B 0,C 180,E1 6624.742,E2 6624.742} C_VEL
LIN {X 0,Y 480.486,Z 580.66,A -85,B 0,C 180,E1 6629.842,E2 6629.842} C_VEL
LIN {X 0,Y 480.645,Z 580.66,A -85,B 0,C 180,E1 6635.918,E2 6635.918} C_VEL
LIN {X 0,Y 480.863,Z 580.66,A -85,B 0,C 180,E1 6641.716,E2 6641.716} C_VEL
LIN {X 0,Y 480.753,Z 580.66,A -85,B 0,C 180,E1 6647.312,E2 6647.312} C_VEL
LIN {X 0,Y 481.101,Z 580.66,A -85,B 0,C 180,E1 6653.011,E2 6653.011} C_VEL
LIN {X 0,Y 481.407,Z 580.66,A -85,B 0,C 180,E1 6658.207,E2 6658.207} C_VEL
LIN {X 0,Y 481.24,Z 580.66,A -85,B 0,C 180,E1 6663.599,E2 6663.599} C_VEL
LIN {X 0,Y 481.084,Z 580.66,A -85,B 0,C 180,E1 6669.026,E2 6669.026} C_VEL
LIN {X 0,Y 480.953,Z 580.66,A -85,B 0,C 180,E1 6674.539,E2 6674.539} C_VEL
LIN {X 0,Y 480.809,Z 580.66,A -85,B 0,C 180,E1 6680.198,E2 6680.198} C_VEL
LIN {X 0,Y 480.636,Z 580.66,A -85,B 0,C 180,E1 6686.076,E2 6686.076} C_VEL
LIN {X 0,Y 480.522,Z 580.66,A -85,B 0,C 180,E1 6692.267,E2 6692.267} C_VEL
LIN {X 0,Y 480.403,Z 580.66,A -85,B 0,C 180,E1 6698.919,E2 6698.919} C_VEL
LIN {X 0,Y 480.42,Z 580.66,A -85,B 0,C 180,E1 6703.746,E2 6703.746} C_VEL
LIN {X 0,Y 480.452,Z 580.66,A -85,B 0,C 180,E1 6709.816,E2 6709.816} C_VEL
LIN {X 0,Y 480.518,Z 580.66,A -85,B 0,C 180,E1 6713.859,E2 6713.859} C_VEL
LIN {X 0,Y 476.537,Z 580.66,A -85,B 0,C 180,E1 6715.193,E2 6715.193} C_VEL
LIN {X 0,Y 472.688,Z 580.66,A -85,B 0,C 180,E1 6716.548,E2 6716.548} C_VEL
LIN {X 0,Y 472.74,Z 580.916,A -85,B 0,C 180,E1 6716.855,E2 6716.855} C_VEL
LIN {X 0,Y 488.067,Z 619.933,A -85,B 0,C 180,E1 6718.515,E2 6718.515} C_VEL
LIN {X 0,Y 487.028,Z 666.326,A -85,B 0,C 180,E1 6719.453,E2 6719.453} C_VEL
LIN {X 0,Y 484.928,Z 703.092,A -85,B 0,C 180,E1 6720.853,E2 6720.853} C_VEL
LIN {X 0,Y 482.449,Z 739.021,A -85,B 0,C 180,E1 6722.96,E2 6722.96} C_VEL
LIN {X 0,Y 479.903,Z 771.649,A -85,B 0,C 180,E1 6725.65,E2 6725.65} C_VEL
LIN {X 0,Y 477.546,Z 801.362,A -85,B 0,C 180,E1 6728.975,E2 6728.975} C_VEL
LIN {X 0,Y 475.717,Z 826.096,A -85,B 0,C 180,E1 6732.705,E2 6732.705} C_VEL
LIN {X 0,Y 474.514,Z 845.732,A -85,B 0,C 180,E1 6736.775,E2 6736.775} C_VEL
LIN {X 0,Y 473.895,Z 858.68,A -85,B 0,C 180,E1 6740.838,E2 6740.838} C_VEL
LIN {X 0,Y 473.635,Z 867.188,A -85,B 0,C 180,E1 6745.43,E2 6745.43} C_VEL
LIN {X 0,Y 473.537,Z 870,A -85,B 0,C 180,E1 6749.998,E2 6749.998} C_VEL
LIN {X 0,Y 473.639,Z 867.194,A -85,B 0,C 180,E1 6754.567,E2 6754.567} C_VEL
LIN {X 0,Y 473.873,Z 858.579,A -85,B 0,C 180,E1 6759.202,E2 6759.202} C_VEL
LIN {X 0,Y 474.41,Z 845.734,A -85,B 0,C 180,E1 6763.223,E2 6763.223} C_VEL
LIN {X 0,Y 475.507,Z 827.991,A -85,B 0,C 180,E1 6766.949,E2 6766.949} C_VEL
LIN {X 0,Y 477.238,Z 804.399,A -85,B 0,C 180,E1 6770.621,E2 6770.621} C_VEL
LIN {X 0,Y 479.625,Z 775.102,A -85,B 0,C 180,E1 6774.016,E2 6774.016} C_VEL
LIN {X 0,Y 482.191,Z 742.553,A -85,B 0,C 180,E1 6776.783,E2 6776.783} C_VEL
LIN {X 0,Y 484.762,Z 706.077,A -85,B 0,C 180,E1 6779.003,E2 6779.003} C_VEL
LIN {X 0,Y 486.909,Z 668.233,A -85,B 0,C 180,E1 6780.494,E2 6780.494} C_VEL
LIN {X 0,Y 487.906,Z 624.449,A -85,B 0,C 180,E1 6781.422,E2 6781.422} C_VEL
LIN {X 0,Y 486.745,Z 616.851,A -85,B 0,C 180,E1 6781.617,E2 6781.617} C_VEL
LIN {X 0,Y 472.712,Z 580.66,A -85,B 0,C 180,E1 6783.208,E2 6783.208} C_VEL
LIN {X 0,Y 472.404,Z 580.66,A -85,B 0,C 180,E1 6789.949,E2 6789.949} C_VEL
LIN {X 0,Y 472.453,Z 580.66,A -85,B 0,C 180,E1 6795.359,E2 6795.359} C_VEL
LIN {X 0,Y 472.557,Z 580.66,A -85,B 0,C 180,E1 6800.309,E2 6800.309} C_VEL
LIN {X 0,Y 472.538,Z 580.66,A -85,B 0,C 180,E1 6806.12,E2 6806.12} C_VEL
LIN {X 0,Y 472.652,Z 580.66,A -85,B 0,C 180,E1 6811.386,E2 6811.386} C_VEL
LIN {X 0,Y 472.837,Z 580.66,A -85,B 0,C 180,E1 6817.732,E2 6817.732} C_VEL
LIN {X 0,Y 472.908,Z 580.66,A -85,B 0,C 180,E1 6823.309,E2 6823.309} C_VEL
LIN {X 0,Y 472.964,Z 580.66,A -85,B 0,C 180,E1 6828.961,E2 6828.961} C_VEL
LIN {X 0,Y 473.245,Z 580.66,A -85,B 0,C 180,E1 6834.508,E2 6834.508} C_VEL
LIN {X 0,Y 473.327,Z 580.66,A -85,B 0,C 180,E1 6839.997,E2 6839.997} C_VEL
LIN {X 0,Y 473.237,Z 580.66,A -85,B 0,C 180,E1 6845.485,E2 6845.485} C_VEL
LIN {X 0,Y 473.066,Z 580.66,A -85,B 0,C 180,E1 6851.029,E2 6851.029} C_VEL
LIN {X 0,Y 472.93,Z 580.66,A -85,B 0,C 180,E1 6856.835,E2 6856.835} C_VEL
LIN {X 0,Y 472.822,Z 580.66,A -85,B 0,C 180,E1 6862.512,E2 6862.512} C_VEL
LIN {X 0,Y 472.627,Z 580.66,A -85,B 0,C 180,E1 6868.608,E2 6868.608} C_VEL
LIN {X 0,Y 472.556,Z 580.66,A -85,B 0,C 180,E1 6875.077,E2 6875.077} C_VEL
LIN {X 0,Y 472.383,Z 580.66,A -85,B 0,C 180,E1 6882.122,E2 6882.122} C_VEL
LIN {X 0,Y 472.503,Z 580.66,A -85,B 0,C 180,E1 6887.887,E2 6887.887} C_VEL
LIN {X 0,Y 472.652,Z 580.66,A -85,B 0,C 180,E1 6892.942,E2 6892.942} C_VEL
LIN {X 0,Y 472.596,Z 580.66,A -85,B 0,C 180,E1 6899.539,E2 6899.539} C_VEL
LIN {X 0,Y 472.661,Z 580.815,A -85,B 0,C 180,E1 6903.455,E2 6903.455} C_VEL
LIN {X 0,Y 483.129,Z 611.289,A -85,B 0,C 180,E1 6905.816,E2 6905.816} C_VEL
LIN {X 0,Y 484.796,Z 620.784,A -85,B 0,C 180,E1 6906.6,E2 6906.6} C_VEL
LIN {X 0,Y 482.295,Z 648.578,A -85,B 0,C 180,E1 6908.914,E2 6908.914} C_VEL
LIN {X 0,Y 479.516,Z 673.777,A -85,B 0,C 180,E1 6911.898,E2 6911.898} C_VEL
LIN {X 0,Y 477.211,Z 694.463,A -85,B 0,C 180,E1 6915.349,E2 6915.349} C_VEL
LIN {X 0,Y 475.416,Z 711.042,A -85,B 0,C 180,E1 6919.392,E2 6919.392} C_VEL
LIN {X 0,Y 474.498,Z 721.716,A -85,B 0,C 180,E1 6923.611,E2 6923.611} C_VEL
LIN {X 0,Y 474.291,Z 725.683,A -85,B 0,C 180,E1 6926.353,E2 6926.353} C_VEL
LIN {X 0,Y 474.106,Z 727.532,A -85,B 0,C 180,E1 6930.002,E2 6930.002} C_VEL
LIN {X 0,Y 474.409,Z 724.475,A -85,B 0,C 180,E1 6934.562,E2 6934.562} C_VEL
LIN {X 0,Y 475.012,Z 716.383,A -85,B 0,C 180,E1 6938.68,E2 6938.68} C_VEL
LIN {X 0,Y 476.407,Z 702.458,A -85,B 0,C 180,E1 6942.811,E2 6942.811} C_VEL
LIN {X 0,Y 478.415,Z 683.781,A -85,B 0,C 180,E1 6946.492,E2 6946.492} C_VEL
LIN {X 0,Y 480.967,Z 660.925,A -85,B 0,C 180,E1 6949.658,E2 6949.658} C_VEL
LIN {X 0,Y 483.612,Z 634.513,A -85,B 0,C 180,E1 6952.274,E2 6952.274} C_VEL
LIN {X 0,Y 484.287,Z 614.945,A -85,B 0,C 180,E1 6953.763,E2 6953.763} C_VEL
LIN {X 0,Y 474.329,Z 586.13,A -85,B 0,C 180,E1 6956.103,E2 6956.103} C_VEL
LIN {X 0,Y 472.638,Z 580.66,A -85,B 0,C 180,E1 6956.55,E2 6956.55} C_VEL
LIN {X 0,Y 472.503,Z 580.66,A -85,B 0,C 180,E1 6962.882,E2 6962.882} C_VEL
LIN {X 0,Y 472.627,Z 580.66,A -85,B 0,C 180,E1 6967.346,E2 6967.346} C_VEL
LIN {X 0,Y 472.444,Z 580.66,A -85,B 0,C 180,E1 6972.735,E2 6972.735} C_VEL
LIN {X 0,Y 472.461,Z 580.66,A -85,B 0,C 180,E1 6977.887,E2 6977.887} C_VEL
LIN {X 0,Y 472.607,Z 580.66,A -85,B 0,C 180,E1 6982.96,E2 6982.96} C_VEL
LIN {X 0,Y 472.558,Z 580.66,A -85,B 0,C 180,E1 6989.56,E2 6989.56} C_VEL
LIN {X 0,Y 472.733,Z 580.66,A -85,B 0,C 180,E1 6995.489,E2 6995.489} C_VEL
LIN {X 0,Y 472.936,Z 580.66,A -85,B 0,C 180,E1 7001.399,E2 7001.399} C_VEL
LIN {X 0,Y 472.836,Z 580.66,A -85,B 0,C 180,E1 7007.096,E2 7007.096} C_VEL
LIN {X 0,Y 473.17,Z 580.66,A -85,B 0,C 180,E1 7013.006,E2 7013.006} C_VEL
LIN {X 0,Y 473.496,Z 580.66,A -85,B 0,C 180,E1 7018.177,E2 7018.177} C_VEL
LIN {X 0,Y 473.329,Z 580.66,A -85,B 0,C 180,E1 7023.659,E2 7023.659} C_VEL
LIN {X 0,Y 473.187,Z 580.66,A -85,B 0,C 180,E1 7029.178,E2 7029.178} C_VEL
LIN {X 0,Y 473.013,Z 580.66,A -85,B 0,C 180,E1 7034.788,E2 7034.788} C_VEL
LIN {X 0,Y 472.861,Z 580.66,A -85,B 0,C 180,E1 7040.552,E2 7040.552} C_VEL
LIN {X 0,Y 472.684,Z 580.66,A -85,B 0,C 180,E1 7046.639,E2 7046.639} C_VEL
LIN {X 0,Y 472.535,Z 580.66,A -85,B 0,C 180,E1 7052.881,E2 7052.881} C_VEL
LIN {X 0,Y 472.517,Z 580.66,A -85,B 0,C 180,E1 7057.357,E2 7057.357} C_VEL
LIN {X 0,Y 472.433,Z 580.66,A -85,B 0,C 180,E1 7062.724,E2 7062.724} C_VEL
LIN {X 0,Y 472.489,Z 580.66,A -85,B 0,C 180,E1 7067.881,E2 7067.881} C_VEL
LIN {X 0,Y 472.567,Z 580.66,A -85,B 0,C 180,E1 7073.856,E2 7073.856} C_VEL
LIN {X 0,Y 472.688,Z 580.66,A -85,B 0,C 180,E1 7076.548,E2 7076.548} C_VEL
LIN {X 0,Y 474.559,Z 583.562,A -85,B 0,C 180,E1 7077.016,E2 7077.016} C_VEL
LIN {X 0,Y 476.904,Z 594.699,A -85,B 0,C 180,E1 7077.368,E2 7077.368} C_VEL
LIN {X 0,Y 477.202,Z 612.785,A -85,B 0,C 180,E1 7077.726,E2 7077.726} C_VEL
LIN {X 0,Y 477.573,Z 613.967,A -85,B 0,C 180,E1 7077.772,E2 7077.772} C_VEL
LIN {X 0,Y 481.038,Z 623.573,A -85,B 0,C 180,E1 7078.159,E2 7078.159} C_VEL
LIN {X 0,Y 479.778,Z 667.279,A -85,B 0,C 180,E1 7079.101,E2 7079.101} C_VEL
LIN {X 0,Y 477.511,Z 703.725,A -85,B 0,C 180,E1 7080.544,E2 7080.544} C_VEL
LIN {X 0,Y 474.785,Z 740.341,A -85,B 0,C 180,E1 7082.779,E2 7082.779} C_VEL
LIN {X 0,Y 472.08,Z 773.123,A -85,B 0,C 180,E1 7085.582,E2 7085.582} C_VEL
LIN {X 0,Y 469.655,Z 802.379,A -85,B 0,C 180,E1 7088.975,E2 7088.975} C_VEL
LIN {X 0,Y 467.786,Z 826.703,A -85,B 0,C 180,E1 7092.797,E2 7092.797} C_VEL
LIN {X 0,Y 466.583,Z 845.805,A -85,B 0,C 180,E1 7096.914,E2 7096.914} C_VEL
LIN {X 0,Y 465.973,Z 859.402,A -85,B 0,C 180,E1 7101.19,E2 7101.19} C_VEL
LIN {X 0,Y 465.742,Z 867.134,A -85,B 0,C 180,E1 7105.353,E2 7105.353} C_VEL
LIN {X 0,Y 465.647,Z 869.998,A -85,B 0,C 180,E1 7109.998,E2 7109.998} C_VEL
LIN {X 0,Y 465.768,Z 868.152,A -85,B 0,C 180,E1 7113.713,E2 7113.713} C_VEL
LIN {X 0,Y 465.965,Z 860.682,A -85,B 0,C 180,E1 7118.282,E2 7118.282} C_VEL
LIN {X 0,Y 466.411,Z 847.647,A -85,B 0,C 180,E1 7122.612,E2 7122.612} C_VEL
LIN {X 0,Y 467.49,Z 829.72,A -85,B 0,C 180,E1 7126.644,E2 7126.644} C_VEL
LIN {X 0,Y 469.249,Z 806.375,A -85,B 0,C 180,E1 7130.467,E2 7130.467} C_VEL
LIN {X 0,Y 471.638,Z 778.07,A -85,B 0,C 180,E1 7133.911,E2 7133.911} C_VEL
LIN {X 0,Y 474.435,Z 745.016,A -85,B 0,C 180,E1 7136.877,E2 7136.877} C_VEL
LIN {X 0,Y 477,Z 710.423,A -85,B 0,C 180,E1 7139.105,E2 7139.105} C_VEL
LIN {X 0,Y 479.339,Z 673.65,A -85,B 0,C 180,E1 7140.7,E2 7140.7} C_VEL
LIN {X 0,Y 480.787,Z 633.548,A -85,B 0,C 180,E1 7141.682,E2 7141.682} C_VEL
LIN {X 0,Y 479.968,Z 619.707,A -85,B 0,C 180,E1 7141.975,E2 7141.975} C_VEL
LIN {X 0,Y 464.739,Z 580.66,A -85,B 0,C 180,E1 7143.746,E2 7143.746} C_VEL
LIN {X 0,Y 464.452,Z 580.66,A -85,B 0,C 180,E1 7150.522,E2 7150.522} C_VEL
LIN {X 0,Y 464.578,Z 580.66,A -85,B 0,C 180,E1 7156.992,E2 7156.992} C_VEL
LIN {X 0,Y 464.621,Z 580.66,A -85,B 0,C 180,E1 7161.896,E2 7161.896} C_VEL
LIN {X 0,Y 464.619,Z 580.66,A -85,B 0,C 180,E1 7168.69,E2 7168.69} C_VEL
LIN {X 0,Y 464.848,Z 580.66,A -85,B 0,C 180,E1 7175.349,E2 7175.349} C_VEL
LIN {X 0,Y 464.994,Z 580.66,A -85,B 0,C 180,E1 7181.062,E2 7181.062} C_VEL
LIN {X 0,Y 465.002,Z 580.66,A -85,B 0,C 180,E1 7186.868,E2 7186.868} C_VEL
LIN {X 0,Y 465.276,Z 580.66,A -85,B 0,C 180,E1 7192.543,E2 7192.543} C_VEL
LIN {X 0,Y 465.567,Z 580.66,A -85,B 0,C 180,E1 7198.139,E2 7198.139} C_VEL
LIN {X 0,Y 465.525,Z 580.66,A -85,B 0,C 180,E1 7203.713,E2 7203.713} C_VEL
LIN {X 0,Y 465.226,Z 580.66,A -85,B 0,C 180,E1 7209.329,E2 7209.329} C_VEL
LIN {X 0,Y 465.087,Z 580.66,A -85,B 0,C 180,E1 7215.039,E2 7215.039} C_VEL
LIN {X 0,Y 464.929,Z 580.66,A -85,B 0,C 180,E1 7220.912,E2 7220.912} C_VEL
LIN {X 0,Y 464.729,Z 580.66,A -85,B 0,C 180,E1 7227.032,E2 7227.032} C_VEL
LIN {X 0,Y 464.626,Z 580.66,A -85,B 0,C 180,E1 7233.505,E2 7233.505} C_VEL
LIN {X 0,Y 464.44,Z 580.66,A -85,B 0,C 180,E1 7240.518,E2 7240.518} C_VEL
LIN {X 0,Y 464.59,Z 580.66,A -85,B 0,C 180,E1 7246.998,E2 7246.998} C_VEL
LIN {X 0,Y 464.613,Z 580.66,A -85,B 0,C 180,E1 7251.9,E2 7251.9} C_VEL
LIN {X 0,Y 464.585,Z 580.66,A -85,B 0,C 180,E1 7258.692,E2 7258.692} C_VEL
LIN {X 0,Y 464.71,Z 580.66,A -85,B 0,C 180,E1 7262.854,E2 7262.854} C_VEL
LIN {X 0,Y 475.112,Z 610.826,A -85,B 0,C 180,E1 7265.217,E2 7265.217} C_VEL
LIN {X 0,Y 477.687,Z 622.657,A -85,B 0,C 180,E1 7266.249,E2 7266.249} C_VEL
LIN {X 0,Y 474.926,Z 651.199,A -85,B 0,C 180,E1 7268.693,E2 7268.693} C_VEL
LIN {X 0,Y 472.13,Z 675.157,A -85,B 0,C 180,E1 7271.604,E2 7271.604} C_VEL
LIN {X 0,Y 469.665,Z 695.773,A -85,B 0,C 180,E1 7275.108,E2 7275.108} C_VEL
LIN {X 0,Y 467.928,Z 711.037,A -85,B 0,C 180,E1 7278.846,E2 7278.846} C_VEL
LIN {X 0,Y 466.906,Z 721.143,A -85,B 0,C 180,E1 7282.574,E2 7282.574} C_VEL
LIN {X 0,Y 466.495,Z 726.882,A -85,B 0,C 180,E1 7286.292,E2 7286.292} C_VEL
LIN {X 0,Y 466.297,Z 728.718,A -85,B 0,C 180,E1 7290.002,E2 7290.002} C_VEL
LIN {X 0,Y 466.636,Z 725.679,A -85,B 0,C 180,E1 7294.638,E2 7294.638} C_VEL
LIN {X 0,Y 467.288,Z 717.632,A -85,B 0,C 180,E1 7298.825,E2 7298.825} C_VEL
LIN {X 0,Y 468.801,Z 703.76,A -85,B 0,C 180,E1 7303.023,E2 7303.023} C_VEL
LIN {X 0,Y 470.96,Z 685.128,A -85,B 0,C 180,E1 7306.761,E2 7306.761} C_VEL
LIN {X 0,Y 473.668,Z 662.359,A -85,B 0,C 180,E1 7309.973,E2 7309.973} C_VEL
LIN {X 0,Y 476.583,Z 635.044,A -85,B 0,C 180,E1 7312.712,E2 7312.712} C_VEL
LIN {X 0,Y 477.417,Z 618.133,A -85,B 0,C 180,E1 7314.022,E2 7314.022} C_VEL
LIN {X 0,Y 467.207,Z 588.308,A -85,B 0,C 180,E1 7316.524,E2 7316.524} C_VEL
LIN {X 0,Y 464.689,Z 580.66,A -85,B 0,C 180,E1 7317.141,E2 7317.141} C_VEL
LIN {X 0,Y 464.599,Z 580.66,A -85,B 0,C 180,E1 7323.515,E2 7323.515} C_VEL
LIN {X 0,Y 464.584,Z 580.66,A -85,B 0,C 180,E1 7328.794,E2 7328.794} C_VEL
LIN {X 0,Y 464.519,Z 580.66,A -85,B 0,C 180,E1 7335.616,E2 7335.616} C_VEL
LIN {X 0,Y 464.598,Z 580.66,A -85,B 0,C 180,E1 7341.903,E2 7341.903} C_VEL
LIN {X 0,Y 464.582,Z 580.66,A -85,B 0,C 180,E1 7348.696,E2 7348.696} C_VEL
LIN {X 0,Y 464.816,Z 580.66,A -85,B 0,C 180,E1 7355.365,E2 7355.365} C_VEL
LIN {X 0,Y 464.987,Z 580.66,A -85,B 0,C 180,E1 7361.069,E2 7361.069} C_VEL
LIN {X 0,Y 464.912,Z 580.66,A -85,B 0,C 180,E1 7366.872,E2 7366.872} C_VEL
LIN {X 0,Y 465.263,Z 580.66,A -85,B 0,C 180,E1 7373.003,E2 7373.003} C_VEL
LIN {X 0,Y 465.594,Z 580.66,A -85,B 0,C 180,E1 7378.146,E2 7378.146} C_VEL
LIN {X 0,Y 465.433,Z 580.66,A -85,B 0,C 180,E1 7383.721,E2 7383.721} C_VEL
LIN {X 0,Y 465.26,Z 580.66,A -85,B 0,C 180,E1 7389.335,E2 7389.335} C_VEL
LIN {X 0,Y 465.072,Z 580.66,A -85,B 0,C 180,E1 7395.047,E2 7395.047} C_VEL
LIN {X 0,Y 464.944,Z 580.66,A -85,B 0,C 180,E1 7400.918,E2 7400.918} C_VEL
LIN {X 0,Y 464.751,Z 580.66,A -85,B 0,C 180,E1 7407.038,E2 7407.038} C_VEL
LIN {X 0,Y 464.617,Z 580.66,A -85,B 0,C 180,E1 7413.514,E2 7413.514} C_VEL
LIN {X 0,Y 464.467,Z 580.66,A -85,B 0,C 180,E1 7420.525,E2 7420.525} C_VEL
LIN {X 0,Y 464.58,Z 580.66,A -85,B 0,C 180,E1 7426.993,E2 7426.993} C_VEL
LIN {X 0,Y 464.635,Z 580.66,A -85,B 0,C 180,E1 7431.898,E2 7431.898} C_VEL
LIN {X 0,Y 464.758,Z 580.66,A -85,B 0,C 180,E1 7436.257,E2 7436.257} C_VEL
LIN {X 0,Y 477.573,Z 613.967,A -85,B 0,C 180,E1 7437.772,E2 7437.772} C_VEL
LIN {X 0,Y 477.527,Z 622.502,A -85,B 0,C 180,E1 7437.917,E2 7437.917} C_VEL
LIN {X 0,Y 473.829,Z 637.319,A -85,B 0,C 180,E1 7437.956,E2 7437.956} C_VEL
LIN {X 0,Y 471.97,Z 676.425,A -85,B 0,C 180,E1 7439,E2 7439} C_VEL
LIN {X 0,Y 469.3,Z 714.507,A -85,B 0,C 180,E1 7440.781,E2 7440.781} C_VEL
LIN {X 0,Y 466.434,Z 749.384,A -85,B 0,C 180,E1 7443.198,E2 7443.198} C_VEL
LIN {X 0,Y 463.664,Z 781.431,A -85,B 0,C 180,E1 7446.256,E2 7446.256} C_VEL
LIN {X 0,Y 461.232,Z 809.681,A -85,B 0,C 180,E1 7449.908,E2 7449.908} C_VEL
LIN {X 0,Y 459.54,Z 831.848,A -85,B 0,C 180,E1 7453.792,E2 7453.792} C_VEL
LIN {X 0,Y 458.449,Z 849.621,A -85,B 0,C 180,E1 7458.127,E2 7458.127} C_VEL
LIN {X 0,Y 458.012,Z 861.281,A -85,B 0,C 180,E1 7462.426,E2 7462.426} C_VEL
LIN {X 0,Y 457.918,Z 867.129,A -85,B 0,C 180,E1 7466.22,E2 7466.22} C_VEL
LIN {X 0,Y 457.826,Z 869.102,A -85,B 0,C 180,E1 7469.998,E2 7469.998} C_VEL
LIN {X 0,Y 457.942,Z 867.135,A -85,B 0,C 180,E1 7473.777,E2 7473.777} C_VEL
LIN {X 0,Y 458.102,Z 859.929,A -85,B 0,C 180,E1 7478.192,E2 7478.192} C_VEL
LIN {X 0,Y 458.508,Z 847.959,A -85,B 0,C 180,E1 7482.35,E2 7482.35} C_VEL
LIN {X 0,Y 459.603,Z 829.495,A -85,B 0,C 180,E1 7486.693,E2 7486.693} C_VEL
LIN {X 0,Y 461.414,Z 806.37,A -85,B 0,C 180,E1 7490.58,E2 7490.58} C_VEL
LIN {X 0,Y 463.911,Z 778.036,A -85,B 0,C 180,E1 7494.111,E2 7494.111} C_VEL
LIN {X 0,Y 466.885,Z 744.784,A -85,B 0,C 180,E1 7497.174,E2 7497.174} C_VEL
LIN {X 0,Y 469.767,Z 708.615,A -85,B 0,C 180,E1 7499.542,E2 7499.542} C_VEL
LIN {X 0,Y 472.404,Z 670.673,A -85,B 0,C 180,E1 7501.201,E2 7501.201} C_VEL
LIN {X 0,Y 473.81,Z 628.629,A -85,B 0,C 180,E1 7502.208,E2 7502.208} C_VEL
LIN {X 0,Y 472.759,Z 621.536,A -85,B 0,C 180,E1 7502.404,E2 7502.404} C_VEL
LIN {X 0,Y 456.811,Z 580.66,A -85,B 0,C 180,E1 7504.328,E2 7504.328} C_VEL
LIN {X 0,Y 456.572,Z 580.66,A -85,B 0,C 180,E1 7511.372,E2 7511.372} C_VEL
LIN {X 0,Y 456.668,Z 580.66,A -85,B 0,C 180,E1 7516.627,E2 7516.627} C_VEL
LIN {X 0,Y 456.68,Z 580.66,A -85,B 0,C 180,E1 7522.463,E2 7522.463} C_VEL
LIN {X 0,Y 456.682,Z 580.66,A -85,B 0,C 180,E1 7529.208,E2 7529.208} C_VEL
LIN {X 0,Y 456.827,Z 580.66,A -85,B 0,C 180,E1 7534.568,E2 7534.568} C_VEL
LIN {X 0,Y 457.065,Z 580.66,A -85,B 0,C 180,E1 7540.72,E2 7540.72} C_VEL
LIN {X 0,Y 457.065,Z 580.66,A -85,B 0,C 180,E1 7546.635,E2 7546.635} C_VEL
LIN {X 0,Y 457.347,Z 580.66,A -85,B 0,C 180,E1 7552.413,E2 7552.413} C_VEL
LIN {X 0,Y 457.657,Z 580.66,A -85,B 0,C 180,E1 7558.107,E2 7558.107} C_VEL
LIN {X 0,Y 457.608,Z 580.66,A -85,B 0,C 180,E1 7563.778,E2 7563.778} C_VEL
LIN {X 0,Y 457.302,Z 580.66,A -85,B 0,C 180,E1 7569.492,E2 7569.492} C_VEL
LIN {X 0,Y 457.147,Z 580.66,A -85,B 0,C 180,E1 7575.307,E2 7575.307} C_VEL
LIN {X 0,Y 456.972,Z 580.66,A -85,B 0,C 180,E1 7581.293,E2 7581.293} C_VEL
LIN {X 0,Y 456.788,Z 580.66,A -85,B 0,C 180,E1 7587.541,E2 7587.541} C_VEL
LIN {X 0,Y 456.634,Z 580.66,A -85,B 0,C 180,E1 7594.302,E2 7594.302} C_VEL
LIN {X 0,Y 456.553,Z 580.66,A -85,B 0,C 180,E1 7600.525,E2 7600.525} C_VEL
LIN {X 0,Y 456.671,Z 580.66,A -85,B 0,C 180,E1 7606.621,E2 7606.621} C_VEL
LIN {X 0,Y 456.671,Z 580.66,A -85,B 0,C 180,E1 7612.458,E2 7612.458} C_VEL
LIN {X 0,Y 456.648,Z 580.66,A -85,B 0,C 180,E1 7619.208,E2 7619.208} C_VEL
LIN {X 0,Y 456.842,Z 581.236,A -85,B 0,C 180,E1 7622.275,E2 7622.275} C_VEL
LIN {X 0,Y 467.758,Z 612.412,A -85,B 0,C 180,E1 7624.79,E2 7624.79} C_VEL
LIN {X 0,Y 470.545,Z 625.146,A -85,B 0,C 180,E1 7625.934,E2 7625.934} C_VEL
LIN {X 0,Y 467.553,Z 653.72,A -85,B 0,C 180,E1 7628.465,E2 7628.465} C_VEL
LIN {X 0,Y 464.586,Z 678.147,A -85,B 0,C 180,E1 7631.54,E2 7631.54} C_VEL
LIN {X 0,Y 461.949,Z 698.178,A -85,B 0,C 180,E1 7635.096,E2 7635.096} C_VEL
LIN {X 0,Y 460.074,Z 713.617,A -85,B 0,C 180,E1 7639.053,E2 7639.053} C_VEL
LIN {X 0,Y 458.981,Z 724.148,A -85,B 0,C 180,E1 7643.394,E2 7643.394} C_VEL
LIN {X 0,Y 458.717,Z 728.075,A -85,B 0,C 180,E1 7646.229,E2 7646.229} C_VEL
LIN {X 0,Y 458.487,Z 729.905,A -85,B 0,C 180,E1 7650.002,E2 7650.002} C_VEL
LIN {X 0,Y 458.848,Z 726.878,A -85,B 0,C 180,E1 7654.717,E2 7654.717} C_VEL
LIN {X 0,Y 459.564,Z 718.865,A -85,B 0,C 180,E1 7658.974,E2 7658.974} C_VEL
LIN {X 0,Y 461.203,Z 705.039,A -85,B 0,C 180,E1 7663.241,E2 7663.241} C_VEL
LIN {X 0,Y 463.497,Z 686.453,A -85,B 0,C 180,E1 7667.039,E2 7667.039} C_VEL
LIN {X 0,Y 466.439,Z 663.222,A -85,B 0,C 180,E1 7670.364,E2 7670.364} C_VEL
LIN {X 0,Y 469.461,Z 636.556,A -85,B 0,C 180,E1 7673.076,E2 7673.076} C_VEL
LIN {X 0,Y 470.306,Z 620.664,A -85,B 0,C 180,E1 7674.34,E2 7674.34} C_VEL
LIN {X 0,Y 460.441,Z 591.272,A -85,B 0,C 180,E1 7676.895,E2 7676.895} C_VEL
LIN {X 0,Y 456.793,Z 580.66,A -85,B 0,C 180,E1 7677.756,E2 7677.756} C_VEL
LIN {X 0,Y 456.64,Z 580.66,A -85,B 0,C 180,E1 7684.31,E2 7684.31} C_VEL
LIN {X 0,Y 456.651,Z 580.66,A -85,B 0,C 180,E1 7690.544,E2 7690.544} C_VEL
LIN {X 0,Y 456.649,Z 580.66,A -85,B 0,C 180,E1 7696.634,E2 7696.634} C_VEL
LIN {X 0,Y 456.659,Z 580.66,A -85,B 0,C 180,E1 7702.471,E2 7702.471} C_VEL
LIN {X 0,Y 456.636,Z 580.66,A -85,B 0,C 180,E1 7709.224,E2 7709.224} C_VEL
LIN {X 0,Y 456.796,Z 580.66,A -85,B 0,C 180,E1 7714.574,E2 7714.574} C_VEL
LIN {X 0,Y 457.059,Z 580.66,A -85,B 0,C 180,E1 7720.727,E2 7720.727} C_VEL
LIN {X 0,Y 457.017,Z 580.66,A -85,B 0,C 180,E1 7726.641,E2 7726.641} C_VEL
LIN {X 0,Y 457.334,Z 580.66,A -85,B 0,C 180,E1 7733.003,E2 7733.003} C_VEL
LIN {X 0,Y 457.684,Z 580.66,A -85,B 0,C 180,E1 7738.114,E2 7738.114} C_VEL
LIN {X 0,Y 457.521,Z 580.66,A -85,B 0,C 180,E1 7743.785,E2 7743.785} C_VEL
LIN {X 0,Y 457.336,Z 580.66,A -85,B 0,C 180,E1 7749.499,E2 7749.499} C_VEL
LIN {X 0,Y 457.132,Z 580.66,A -85,B 0,C 180,E1 7755.315,E2 7755.315} C_VEL
LIN {X 0,Y 456.982,Z 580.66,A -85,B 0,C 180,E1 7761.3,E2 7761.3} C_VEL
LIN {X 0,Y 456.815,Z 580.66,A -85,B 0,C 180,E1 7767.547,E2 7767.547} C_VEL
LIN {X 0,Y 456.632,Z 580.66,A -85,B 0,C 180,E1 7774.296,E2 7774.296} C_VEL
LIN {X 0,Y 456.582,Z 580.66,A -85,B 0,C 180,E1 7780.524,E2 7780.524} C_VEL
LIN {X 0,Y 456.672,Z 580.66,A -85,B 0,C 180,E1 7786.631,E2 7786.631} C_VEL
LIN {X 0,Y 456.695,Z 580.66,A -85,B 0,C 180,E1 7792.466,E2 7792.466} C_VEL
LIN {X 0,Y 456.836,Z 580.66,A -85,B 0,C 180,E1 7795.704,E2 7795.704} C_VEL
LIN {X 0,Y 474.027,Z 626.052,A -85,B 0,C 180,E1 7797.76,E2 7797.76} C_VEL
LIN {X 0,Y 473.829,Z 637.319,A -85,B 0,C 180,E1 7797.956,E2 7797.956} C_VEL
LIN {X 0,Y 469.764,Z 654.349,A -85,B 0,C 180,E1 7798.107,E2 7798.107} C_VEL
LIN {X 0,Y 465.291,Z 671.125,A -85,B 0,C 180,E1 7798.393,E2 7798.393} C_VEL
LIN {X 0,Y 462.519,Z 707.716,A -85,B 0,C 180,E1 7800.031,E2 7800.031} C_VEL
LIN {X 0,Y 459.326,Z 744.362,A -85,B 0,C 180,E1 7802.498,E2 7802.498} C_VEL
LIN {X 0,Y 456.281,Z 776.885,A -85,B 0,C 180,E1 7805.556,E2 7805.556} C_VEL
LIN {X 0,Y 453.768,Z 804.606,A -85,B 0,C 180,E1 7809.053,E2 7809.053} C_VEL
LIN {X 0,Y 451.814,Z 829.18,A -85,B 0,C 180,E1 7813.257,E2 7813.257} C_VEL
LIN {X 0,Y 450.699,Z 846.617,A -85,B 0,C 180,E1 7817.429,E2 7817.429} C_VEL
LIN {X 0,Y 450.253,Z 858.639,A -85,B 0,C 180,E1 7821.646,E2 7821.646} C_VEL
LIN {X 0,Y 450.092,Z 865.927,A -85,B 0,C 180,E1 7826.154,E2 7826.154} C_VEL
LIN {X 0,Y 450.031,Z 867.918,A -85,B 0,C 180,E1 7829.998,E2 7829.998} C_VEL
LIN {X 0,Y 450.138,Z 865.933,A -85,B 0,C 180,E1 7833.843,E2 7833.843} C_VEL
LIN {X 0,Y 450.247,Z 858.665,A -85,B 0,C 180,E1 7838.336,E2 7838.336} C_VEL
LIN {X 0,Y 450.654,Z 846.613,A -85,B 0,C 180,E1 7842.569,E2 7842.569} C_VEL
LIN {X 0,Y 451.743,Z 829.172,A -85,B 0,C 180,E1 7846.742,E2 7846.742} C_VEL
LIN {X 0,Y 453.569,Z 806.336,A -85,B 0,C 180,E1 7850.698,E2 7850.698} C_VEL
LIN {X 0,Y 456.131,Z 778.425,A -85,B 0,C 180,E1 7854.274,E2 7854.274} C_VEL
LIN {X 0,Y 459.237,Z 745.73,A -85,B 0,C 180,E1 7857.385,E2 7857.385} C_VEL
LIN {X 0,Y 462.359,Z 709.705,A -85,B 0,C 180,E1 7859.859,E2 7859.859} C_VEL
LIN {X 0,Y 465.157,Z 672.505,A -85,B 0,C 180,E1 7861.56,E2 7861.56} C_VEL
LIN {X 0,Y 466.842,Z 633.051,A -85,B 0,C 180,E1 7862.587,E2 7862.587} C_VEL
LIN {X 0,Y 465.999,Z 624.171,A -85,B 0,C 180,E1 7862.808,E2 7862.808} C_VEL
LIN {X 0,Y 448.8,Z 580.66,A -85,B 0,C 180,E1 7864.927,E2 7864.927} C_VEL
LIN {X 0,Y 448.652,Z 580.66,A -85,B 0,C 180,E1 7869.716,E2 7869.716} C_VEL
LIN {X 0,Y 448.641,Z 580.66,A -85,B 0,C 180,E1 7875.063,E2 7875.063} C_VEL
LIN {X 0,Y 448.764,Z 580.66,A -85,B 0,C 180,E1 7880.653,E2 7880.653} C_VEL
LIN {X 0,Y 448.707,Z 580.66,A -85,B 0,C 180,E1 7887.446,E2 7887.446} C_VEL
LIN {X 0,Y 448.919,Z 580.66,A -85,B 0,C 180,E1 7894.087,E2 7894.087} C_VEL
LIN {X 0,Y 449.109,Z 580.66,A -85,B 0,C 180,E1 7900.365,E2 7900.365} C_VEL
LIN {X 0,Y 449.152,Z 580.66,A -85,B 0,C 180,E1 7906.962,E2 7906.962} C_VEL
LIN {X 0,Y 449.432,Z 580.66,A -85,B 0,C 180,E1 7912.279,E2 7912.279} C_VEL
LIN {X 0,Y 449.773,Z 580.66,A -85,B 0,C 180,E1 7918.074,E2 7918.074} C_VEL
LIN {X 0,Y 449.691,Z 580.66,A -85,B 0,C 180,E1 7923.844,E2 7923.844} C_VEL
LIN {X 0,Y 449.374,Z 580.66,A -85,B 0,C 180,E1 7929.661,E2 7929.661} C_VEL
LIN {X 0,Y 449.249,Z 580.66,A -85,B 0,C 180,E1 7935.583,E2 7935.583} C_VEL
LIN {X 0,Y 449.039,Z 580.66,A -85,B 0,C 180,E1 7941.688,E2 7941.688} C_VEL
LIN {X 0,Y 448.809,Z 580.66,A -85,B 0,C 180,E1 7948.074,E2 7948.074} C_VEL
LIN {X 0,Y 448.668,Z 580.66,A -85,B 0,C 180,E1 7954.865,E2 7954.865} C_VEL
LIN {X 0,Y 448.634,Z 580.66,A -85,B 0,C 180,E1 7959.714,E2 7959.714} C_VEL
LIN {X 0,Y 448.65,Z 580.66,A -85,B 0,C 180,E1 7965.069,E2 7965.069} C_VEL
LIN {X 0,Y 448.791,Z 580.66,A -85,B 0,C 180,E1 7970.643,E2 7970.643} C_VEL
LIN {X 0,Y 448.676,Z 580.66,A -85,B 0,C 180,E1 7977.448,E2 7977.448} C_VEL
LIN {X 0,Y 448.934,Z 581.114,A -85,B 0,C 180,E1 7981.637,E2 7981.637} C_VEL
LIN {X 0,Y 459.988,Z 612.673,A -85,B 0,C 180,E1 7984.223,E2 7984.223} C_VEL
LIN {X 0,Y 463.487,Z 626.864,A -85,B 0,C 180,E1 7985.555,E2 7985.555} C_VEL
LIN {X 0,Y 460.341,Z 655.124,A -85,B 0,C 180,E1 7988.11,E2 7988.11} C_VEL
LIN {X 0,Y 457.196,Z 679.485,A -85,B 0,C 180,E1 7991.231,E2 7991.231} C_VEL
LIN {X 0,Y 454.403,Z 699.453,A -85,B 0,C 180,E1 7994.842,E2 7994.842} C_VEL
LIN {X 0,Y 452.325,Z 715.494,A -85,B 0,C 180,E1 7999.087,E2 7999.087} C_VEL
LIN {X 0,Y 451.218,Z 725.355,A -85,B 0,C 180,E1 8003.28,E2 8003.28} C_VEL
LIN {X 0,Y 450.933,Z 729.266,A -85,B 0,C 180,E1 8006.164,E2 8006.164} C_VEL
LIN {X 0,Y 450.688,Z 731.09,A -85,B 0,C 180,E1 8010.002,E2 8010.002} C_VEL
LIN {X 0,Y 451.068,Z 728.074,A -85,B 0,C 180,E1 8014.799,E2 8014.799} C_VEL
LIN {X 0,Y 451.853,Z 720.089,A -85,B 0,C 180,E1 8019.129,E2 8019.129} C_VEL
LIN {X 0,Y 453.599,Z 706.307,A -85,B 0,C 180,E1 8023.467,E2 8023.467} C_VEL
LIN {X 0,Y 456.036,Z 687.763,A -85,B 0,C 180,E1 8027.327,E2 8027.327} C_VEL
LIN {X 0,Y 459.18,Z 664.441,A -85,B 0,C 180,E1 8030.723,E2 8030.723} C_VEL
LIN {X 0,Y 462.398,Z 637.427,A -85,B 0,C 180,E1 8033.508,E2 8033.508} C_VEL
LIN {X 0,Y 463.032,Z 622.609,A -85,B 0,C 180,E1 8034.723,E2 8034.723} C_VEL
LIN {X 0,Y 452.817,Z 592.068,A -85,B 0,C 180,E1 8037.451,E2 8037.451} C_VEL
LIN {X 0,Y 448.913,Z 580.66,A -85,B 0,C 180,E1 8038.319,E2 8038.319} C_VEL
LIN {X 0,Y 448.694,Z 580.66,A -85,B 0,C 180,E1 8044.87,E2 8044.87} C_VEL
LIN {X 0,Y 448.724,Z 580.66,A -85,B 0,C 180,E1 8049.713,E2 8049.713} C_VEL
LIN {X 0,Y 448.648,Z 580.66,A -85,B 0,C 180,E1 8055.074,E2 8055.074} C_VEL
LIN {X 0,Y 448.739,Z 580.66,A -85,B 0,C 180,E1 8060.662,E2 8060.662} C_VEL
LIN {X 0,Y 448.673,Z 580.66,A -85,B 0,C 180,E1 8067.452,E2 8067.452} C_VEL
LIN {X 0,Y 448.881,Z 580.66,A -85,B 0,C 180,E1 8074.093,E2 8074.093} C_VEL
LIN {X 0,Y 449.104,Z 580.66,A -85,B 0,C 180,E1 8080.372,E2 8080.372} C_VEL
LIN {X 0,Y 449.093,Z 580.66,A -85,B 0,C 180,E1 8087.009,E2 8087.009} C_VEL
LIN {X 0,Y 449.428,Z 580.66,A -85,B 0,C 180,E1 8093.006,E2 8093.006} C_VEL
LIN {X 0,Y 449.799,Z 580.66,A -85,B 0,C 180,E1 8098.081,E2 8098.081} C_VEL
LIN {X 0,Y 449.607,Z 580.66,A -85,B 0,C 180,E1 8103.852,E2 8103.852} C_VEL
LIN {X 0,Y 449.408,Z 580.66,A -85,B 0,C 180,E1 8109.668,E2 8109.668} C_VEL
LIN {X 0,Y 449.232,Z 580.66,A -85,B 0,C 180,E1 8115.591,E2 8115.591} C_VEL
LIN {X 0,Y 449.051,Z 580.66,A -85,B 0,C 180,E1 8121.696,E2 8121.696} C_VEL
LIN {X 0,Y 448.833,Z 580.66,A -85,B 0,C 180,E1 8128.08,E2 8128.08} C_VEL
LIN {X 0,Y 448.668,Z 580.66,A -85,B 0,C 180,E1 8134.874,E2 8134.874} C_VEL
LIN {X 0,Y 448.662,Z 580.66,A -85,B 0,C 180,E1 8139.72,E2 8139.72} C_VEL
LIN {X 0,Y 448.649,Z 580.66,A -85,B 0,C 180,E1 8145.065,E2 8145.065} C_VEL
LIN {X 0,Y 448.777,Z 580.66,A -85,B 0,C 180,E1 8150.656,E2 8150.656} C_VEL
LIN {X 0,Y 448.885,Z 581.365,A -85,B 0,C 180,E1 8155.125,E2 8155.125} C_VEL
LIN {X 0,Y 467.02,Z 626.644,A -85,B 0,C 180,E1 8157.308,E2 8157.308} C_VEL
LIN {X 0,Y 465.572,Z 667.28,A -85,B 0,C 180,E1 8158.262,E2 8158.262} C_VEL
LIN {X 0,Y 465.291,Z 671.125,A -85,B 0,C 180,E1 8158.393,E2 8158.393} C_VEL
LIN {X 0,Y 455.9,Z 701.784,A -85,B 0,C 180,E1 8159.307,E2 8159.307} C_VEL
LIN {X 0,Y 455.624,Z 703.756,A -85,B 0,C 180,E1 8159.411,E2 8159.411} C_VEL
LIN {X 0,Y 452.341,Z 739.086,A -85,B 0,C 180,E1 8161.752,E2 8161.752} C_VEL
LIN {X 0,Y 448.968,Z 773.034,A -85,B 0,C 180,E1 8164.906,E2 8164.906} C_VEL
LIN {X 0,Y 446.244,Z 801.233,A -85,B 0,C 180,E1 8168.443,E2 8168.443} C_VEL
LIN {X 0,Y 444.237,Z 825.116,A -85,B 0,C 180,E1 8172.453,E2 8172.453} C_VEL
LIN {X 0,Y 442.984,Z 843.527,A -85,B 0,C 180,E1 8176.706,E2 8176.706} C_VEL
LIN {X 0,Y 442.48,Z 856.313,A -85,B 0,C 180,E1 8181.01,E2 8181.01} C_VEL
LIN {X 0,Y 442.29,Z 863.628,A -85,B 0,C 180,E1 8185.106,E2 8185.106} C_VEL
LIN {X 0,Y 442.22,Z 866.732,A -85,B 0,C 180,E1 8189.998,E2 8189.998} C_VEL
LIN {X 0,Y 442.311,Z 864.731,A -85,B 0,C 180,E1 8193.911,E2 8193.911} C_VEL
LIN {X 0,Y 442.397,Z 857.49,A -85,B 0,C 180,E1 8198.447,E2 8198.447} C_VEL
LIN {X 0,Y 442.823,Z 845.242,A -85,B 0,C 180,E1 8202.795,E2 8202.795} C_VEL
LIN {X 0,Y 443.962,Z 827.633,A -85,B 0,C 180,E1 8207.044,E2 8207.044} C_VEL
LIN {X 0,Y 446.042,Z 803.247,A -85,B 0,C 180,E1 8211.263,E2 8211.263} C_VEL
LIN {X 0,Y 448.815,Z 774.405,A -85,B 0,C 180,E1 8214.941,E2 8214.941} C_VEL
LIN {X 0,Y 452.164,Z 740.739,A -85,B 0,C 180,E1 8218.121,E2 8218.121} C_VEL
LIN {X 0,Y 455.46,Z 705.808,A -85,B 0,C 180,E1 8220.474,E2 8220.474} C_VEL
LIN {X 0,Y 458.433,Z 668.684,A -85,B 0,C 180,E1 8222.137,E2 8222.137} C_VEL
LIN {X 0,Y 459.708,Z 627.924,A -85,B 0,C 180,E1 8223.174,E2 8223.174} C_VEL
LIN {X 0,Y 442.527,Z 585.507,A -85,B 0,C 180,E1 8225.299,E2 8225.299} C_VEL
LIN {X 0,Y 440.844,Z 580.66,A -85,B 0,C 180,E1 8225.58,E2 8225.58} C_VEL
LIN {X 0,Y 440.634,Z 580.66,A -85,B 0,C 180,E1 8231.113,E2 8231.113} C_VEL
LIN {X 0,Y 440.702,Z 580.66,A -85,B 0,C 180,E1 8236.779,E2 8236.779} C_VEL
LIN {X 0,Y 440.799,Z 580.66,A -85,B 0,C 180,E1 8241.96,E2 8241.96} C_VEL
LIN {X 0,Y 440.759,Z 580.66,A -85,B 0,C 180,E1 8246.784,E2 8246.784} C_VEL
LIN {X 0,Y 440.941,Z 580.66,A -85,B 0,C 180,E1 8253.582,E2 8253.582} C_VEL
LIN {X 0,Y 441.176,Z 580.66,A -85,B 0,C 180,E1 8259.997,E2 8259.997} C_VEL
LIN {X 0,Y 441.223,Z 580.66,A -85,B 0,C 180,E1 8266.146,E2 8266.146} C_VEL
LIN {X 0,Y 441.541,Z 580.66,A -85,B 0,C 180,E1 8272.313,E2 8272.313} C_VEL
LIN {X 0,Y 441.861,Z 580.66,A -85,B 0,C 180,E1 8278.039,E2 8278.039} C_VEL
LIN {X 0,Y 441.775,Z 580.66,A -85,B 0,C 180,E1 8283.913,E2 8283.913} C_VEL
LIN {X 0,Y 441.468,Z 580.66,A -85,B 0,C 180,E1 8289.836,E2 8289.836} C_VEL
LIN {X 0,Y 441.298,Z 580.66,A -85,B 0,C 180,E1 8295.871,E2 8295.871} C_VEL
LIN {X 0,Y 441.066,Z 580.66,A -85,B 0,C 180,E1 8302.533,E2 8302.533} C_VEL
LIN {X 0,Y 440.894,Z 580.66,A -85,B 0,C 180,E1 8308.624,E2 8308.624} C_VEL
LIN {X 0,Y 440.742,Z 580.66,A -85,B 0,C 180,E1 8315.586,E2 8315.586} C_VEL
LIN {X 0,Y 440.645,Z 580.66,A -85,B 0,C 180,E1 8321.121,E2 8321.121} C_VEL
LIN {X 0,Y 440.71,Z 580.66,A -85,B 0,C 180,E1 8326.785,E2 8326.785} C_VEL
LIN {X 0,Y 440.803,Z 580.66,A -85,B 0,C 180,E1 8331.966,E2 8331.966} C_VEL
LIN {X 0,Y 440.731,Z 580.66,A -85,B 0,C 180,E1 8336.787,E2 8336.787} C_VEL
LIN {X 0,Y 440.939,Z 580.957,A -85,B 0,C 180,E1 8340.962,E2 8340.962} C_VEL
LIN {X 0,Y 451.883,Z 611.741,A -85,B 0,C 180,E1 8343.534,E2 8343.534} C_VEL
LIN {X 0,Y 456.369,Z 629.083,A -85,B 0,C 180,E1 8345.201,E2 8345.201} C_VEL
LIN {X 0,Y 453.032,Z 657.6,A -85,B 0,C 180,E1 8347.867,E2 8347.867} C_VEL
LIN {X 0,Y 449.619,Z 682.337,A -85,B 0,C 180,E1 8351.156,E2 8351.156} C_VEL
LIN {X 0,Y 446.55,Z 702.941,A -85,B 0,C 180,E1 8355.071,E2 8355.071} C_VEL
LIN {X 0,Y 444.492,Z 717.978,A -85,B 0,C 180,E1 8359.34,E2 8359.34} C_VEL
LIN {X 0,Y 443.451,Z 726.559,A -85,B 0,C 180,E1 8363.162,E2 8363.162} C_VEL
LIN {X 0,Y 443.154,Z 730.455,A -85,B 0,C 180,E1 8366.097,E2 8366.097} C_VEL
LIN {X 0,Y 442.878,Z 732.276,A -85,B 0,C 180,E1 8370.002,E2 8370.002} C_VEL
LIN {X 0,Y 443.282,Z 729.269,A -85,B 0,C 180,E1 8374.883,E2 8374.883} C_VEL
LIN {X 0,Y 444.146,Z 721.307,A -85,B 0,C 180,E1 8379.288,E2 8379.288} C_VEL
LIN {X 0,Y 446.004,Z 707.564,A -85,B 0,C 180,E1 8383.701,E2 8383.701} C_VEL
LIN {X 0,Y 448.587,Z 689.06,A -85,B 0,C 180,E1 8387.624,E2 8387.624} C_VEL
LIN {X 0,Y 451.935,Z 665.777,A -85,B 0,C 180,E1 8391.075,E2 8391.075} C_VEL
LIN {X 0,Y 455.292,Z 638.896,A -85,B 0,C 180,E1 8393.898,E2 8393.898} C_VEL
LIN {X 0,Y 455.846,Z 624.841,A -85,B 0,C 180,E1 8395.088,E2 8395.088} C_VEL
LIN {X 0,Y 446.005,Z 594.949,A -85,B 0,C 180,E1 8397.857,E2 8397.857} C_VEL
LIN {X 0,Y 440.92,Z 580.66,A -85,B 0,C 180,E1 8398.979,E2 8398.979} C_VEL
LIN {X 0,Y 440.789,Z 580.66,A -85,B 0,C 180,E1 8405.59,E2 8405.59} C_VEL
LIN {X 0,Y 440.707,Z 580.66,A -85,B 0,C 180,E1 8411.136,E2 8411.136} C_VEL
LIN {X 0,Y 440.692,Z 580.66,A -85,B 0,C 180,E1 8416.788,E2 8416.788} C_VEL
LIN {X 0,Y 440.784,Z 580.66,A -85,B 0,C 180,E1 8421.968,E2 8421.968} C_VEL
LIN {X 0,Y 440.728,Z 580.66,A -85,B 0,C 180,E1 8426.79,E2 8426.79} C_VEL
LIN {X 0,Y 440.902,Z 580.66,A -85,B 0,C 180,E1 8433.588,E2 8433.588} C_VEL
LIN {X 0,Y 441.172,Z 580.66,A -85,B 0,C 180,E1 8440.004,E2 8440.004} C_VEL
LIN {X 0,Y 441.148,Z 580.66,A -85,B 0,C 180,E1 8446.151,E2 8446.151} C_VEL
LIN {X 0,Y 441.535,Z 580.66,A -85,B 0,C 180,E1 8453.009,E2 8453.009} C_VEL
LIN {X 0,Y 441.888,Z 580.66,A -85,B 0,C 180,E1 8458.047,E2 8458.047} C_VEL
LIN {X 0,Y 441.694,Z 580.66,A -85,B 0,C 180,E1 8463.921,E2 8463.921} C_VEL
LIN {X 0,Y 441.501,Z 580.66,A -85,B 0,C 180,E1 8469.843,E2 8469.843} C_VEL
LIN {X 0,Y 441.283,Z 580.66,A -85,B 0,C 180,E1 8475.879,E2 8475.879} C_VEL
LIN {X 0,Y 441.037,Z 580.66,A -85,B 0,C 180,E1 8482.515,E2 8482.515} C_VEL
LIN {X 0,Y 440.917,Z 580.66,A -85,B 0,C 180,E1 8488.63,E2 8488.63} C_VEL
LIN {X 0,Y 440.748,Z 580.66,A -85,B 0,C 180,E1 8495.594,E2 8495.594} C_VEL
LIN {X 0,Y 440.648,Z 580.66,A -85,B 0,C 180,E1 8501.116,E2 8501.116} C_VEL
LIN {X 0,Y 440.716,Z 580.66,A -85,B 0,C 180,E1 8506.781,E2 8506.781} C_VEL
LIN {X 0,Y 440.817,Z 580.66,A -85,B 0,C 180,E1 8511.963,E2 8511.963} C_VEL
LIN {X 0,Y 440.92,Z 580.66,A -85,B 0,C 180,E1 8514.455,E2 8514.455} C_VEL
LIN {X 0,Y 460.142,Z 629.076,A -85,B 0,C 180,E1 8516.88,E2 8516.88} C_VEL
LIN {X 0,Y 458.354,Z 669.674,A -85,B 0,C 180,E1 8517.899,E2 8517.899} C_VEL
LIN {X 0,Y 455.624,Z 703.756,A -85,B 0,C 180,E1 8519.411,E2 8519.411} C_VEL
LIN {X 0,Y 450.535,Z 719.584,A -85,B 0,C 180,E1 8520.155,E2 8520.155} C_VEL
LIN {X 0,Y 445.4,Z 734.695,A -85,B 0,C 180,E1 8521.046,E2 8521.046} C_VEL
LIN {X 0,Y 441.826,Z 767.999,A -85,B 0,C 180,E1 8524.09,E2 8524.09} C_VEL
LIN {X 0,Y 438.643,Z 798.778,A -85,B 0,C 180,E1 8527.94,E2 8527.94} C_VEL
LIN {X 0,Y 436.428,Z 823.526,A -85,B 0,C 180,E1 8532.129,E2 8532.129} C_VEL
LIN {X 0,Y 435.148,Z 842.526,A -85,B 0,C 180,E1 8536.575,E2 8536.575} C_VEL
LIN {X 0,Y 434.617,Z 856.18,A -85,B 0,C 180,E1 8541.375,E2 8541.375} C_VEL
LIN {X 0,Y 434.454,Z 863.519,A -85,B 0,C 180,E1 8546.015,E2 8546.015} C_VEL
LIN {X 0,Y 434.409,Z 865.545,A -85,B 0,C 180,E1 8549.998,E2 8549.998} C_VEL
LIN {X 0,Y 434.489,Z 863.526,A -85,B 0,C 180,E1 8553.981,E2 8553.981} C_VEL
LIN {X 0,Y 434.58,Z 856.215,A -85,B 0,C 180,E1 8558.6,E2 8558.6} C_VEL
LIN {X 0,Y 435.071,Z 842.614,A -85,B 0,C 180,E1 8563.399,E2 8563.399} C_VEL
LIN {X 0,Y 436.418,Z 823.53,A -85,B 0,C 180,E1 8567.868,E2 8567.868} C_VEL
LIN {X 0,Y 438.604,Z 798.827,A -85,B 0,C 180,E1 8572.053,E2 8572.053} C_VEL
LIN {X 0,Y 441.662,Z 769.354,A -85,B 0,C 180,E1 8575.769,E2 8575.769} C_VEL
LIN {X 0,Y 445.267,Z 735.746,A -85,B 0,C 180,E1 8578.873,E2 8578.873} C_VEL
LIN {X 0,Y 448.878,Z 699.41,A -85,B 0,C 180,E1 8581.252,E2 8581.252} C_VEL
LIN {X 0,Y 451.824,Z 662.889,A -85,B 0,C 180,E1 8582.79,E2 8582.79} C_VEL
LIN {X 0,Y 452.618,Z 629.621,A -85,B 0,C 180,E1 8583.651,E2 8583.651} C_VEL
LIN {X 0,Y 436.443,Z 589.66,A -85,B 0,C 180,E1 8585.711,E2 8585.711} C_VEL
LIN {X 0,Y 432.843,Z 580.66,A -85,B 0,C 180,E1 8586.258,E2 8586.258} C_VEL
LIN {X 0,Y 432.69,Z 580.66,A -85,B 0,C 180,E1 8592.915,E2 8592.915} C_VEL
LIN {X 0,Y 432.796,Z 580.66,A -85,B 0,C 180,E1 8598.512,E2 8598.512} C_VEL
LIN {X 0,Y 432.819,Z 580.66,A -85,B 0,C 180,E1 8603.651,E2 8603.651} C_VEL
LIN {X 0,Y 432.825,Z 580.66,A -85,B 0,C 180,E1 8608.468,E2 8608.468} C_VEL
LIN {X 0,Y 433.042,Z 580.66,A -85,B 0,C 180,E1 8615.28,E2 8615.28} C_VEL
LIN {X 0,Y 433.266,Z 580.66,A -85,B 0,C 180,E1 8621.73,E2 8621.73} C_VEL
LIN {X 0,Y 433.338,Z 580.66,A -85,B 0,C 180,E1 8627.937,E2 8627.937} C_VEL
LIN {X 0,Y 433.719,Z 580.66,A -85,B 0,C 180,E1 8634.006,E2 8634.006} C_VEL
LIN {X 0,Y 433.869,Z 580.66,A -85,B 0,C 180,E1 8639.996,E2 8639.996} C_VEL
LIN {X 0,Y 433.708,Z 580.66,A -85,B 0,C 180,E1 8645.987,E2 8645.987} C_VEL
LIN {X 0,Y 433.419,Z 580.66,A -85,B 0,C 180,E1 8652.898,E2 8652.898} C_VEL
LIN {X 0,Y 433.263,Z 580.66,A -85,B 0,C 180,E1 8658.262,E2 8658.262} C_VEL
LIN {X 0,Y 433.037,Z 580.66,A -85,B 0,C 180,E1 8665.05,E2 8665.05} C_VEL
LIN {X 0,Y 432.844,Z 580.66,A -85,B 0,C 180,E1 8671.522,E2 8671.522} C_VEL
LIN {X 0,Y 432.757,Z 580.66,A -85,B 0,C 180,E1 8676.686,E2 8676.686} C_VEL
LIN {X 0,Y 432.742,Z 580.66,A -85,B 0,C 180,E1 8682.928,E2 8682.928} C_VEL
LIN {X 0,Y 432.816,Z 580.66,A -85,B 0,C 180,E1 8688.52,E2 8688.52} C_VEL
LIN {X 0,Y 432.809,Z 580.66,A -85,B 0,C 180,E1 8693.655,E2 8693.655} C_VEL
LIN {X 0,Y 432.948,Z 580.789,A -85,B 0,C 180,E1 8700.259,E2 8700.259} C_VEL
LIN {X 0,Y 443.998,Z 611.388,A -85,B 0,C 180,E1 8702.876,E2 8702.876} C_VEL
LIN {X 0,Y 449.285,Z 631.461,A -85,B 0,C 180,E1 8704.857,E2 8704.857} C_VEL
LIN {X 0,Y 445.685,Z 660.072,A -85,B 0,C 180,E1 8707.614,E2 8707.614} C_VEL
LIN {X 0,Y 442.234,Z 683.634,A -85,B 0,C 180,E1 8710.83,E2 8710.83} C_VEL
LIN {X 0,Y 438.997,Z 704.2,A -85,B 0,C 180,E1 8714.808,E2 8714.808} C_VEL
LIN {X 0,Y 436.853,Z 718.918,A -85,B 0,C 180,E1 8719.05,E2 8719.05} C_VEL
LIN {X 0,Y 435.693,Z 727.759,A -85,B 0,C 180,E1 8723.04,E2 8723.04} C_VEL
LIN {X 0,Y 435.375,Z 731.643,A -85,B 0,C 180,E1 8726.027,E2 8726.027} C_VEL
LIN {X 0,Y 435.079,Z 733.461,A -85,B 0,C 180,E1 8730.002,E2 8730.002} C_VEL
LIN {X 0,Y 435.509,Z 730.461,A -85,B 0,C 180,E1 8734.971,E2 8734.971} C_VEL
LIN {X 0,Y 436.424,Z 722.601,A -85,B 0,C 180,E1 8739.421,E2 8739.421} C_VEL
LIN {X 0,Y 438.398,Z 708.817,A -85,B 0,C 180,E1 8743.943,E2 8743.943} C_VEL
LIN {X 0,Y 441.172,Z 690.343,A -85,B 0,C 180,E1 8747.93,E2 8747.93} C_VEL
LIN {X 0,Y 444.692,Z 667.012,A -85,B 0,C 180,E1 8751.452,E2 8751.452} C_VEL
LIN {X 0,Y 448.319,Z 639.533,A -85,B 0,C 180,E1 8754.374,E2 8754.374} C_VEL
LIN {X 0,Y 448.823,Z 627.484,A -85,B 0,C 180,E1 8755.418,E2 8755.418} C_VEL
LIN {X 0,Y 439.11,Z 597.281,A -85,B 0,C 180,E1 8758.312,E2 8758.312} C_VEL
LIN {X 0,Y 432.971,Z 580.66,A -85,B 0,C 180,E1 8759.668,E2 8759.668} C_VEL
LIN {X 0,Y 432.81,Z 580.66,A -85,B 0,C 180,E1 8766.702,E2 8766.702} C_VEL
LIN {X 0,Y 432.774,Z 580.66,A -85,B 0,C 180,E1 8772.938,E2 8772.938} C_VEL
LIN {X 0,Y 432.776,Z 580.66,A -85,B 0,C 180,E1 8778.52,E2 8778.52} C_VEL
LIN {X 0,Y 432.799,Z 580.66,A -85,B 0,C 180,E1 8783.658,E2 8783.658} C_VEL
LIN {X 0,Y 432.784,Z 580.66,A -85,B 0,C 180,E1 8788.473,E2 8788.473} C_VEL
LIN {X 0,Y 433.012,Z 580.66,A -85,B 0,C 180,E1 8795.286,E2 8795.286} C_VEL
LIN {X 0,Y 433.258,Z 580.66,A -85,B 0,C 180,E1 8801.738,E2 8801.738} C_VEL
LIN {X 0,Y 433.294,Z 580.66,A -85,B 0,C 180,E1 8807.944,E2 8807.944} C_VEL
LIN {X 0,Y 433.736,Z 580.66,A -85,B 0,C 180,E1 8814.013,E2 8814.013} C_VEL
LIN {X 0,Y 433.885,Z 580.66,A -85,B 0,C 180,E1 8820.004,E2 8820.004} C_VEL
LIN {X 0,Y 433.692,Z 580.66,A -85,B 0,C 180,E1 8825.995,E2 8825.995} C_VEL
LIN {X 0,Y 433.441,Z 580.66,A -85,B 0,C 180,E1 8832.895,E2 8832.895} C_VEL
LIN {X 0,Y 433.26,Z 580.66,A -85,B 0,C 180,E1 8838.27,E2 8838.27} C_VEL
LIN {X 0,Y 433.006,Z 580.66,A -85,B 0,C 180,E1 8845.033,E2 8845.033} C_VEL
LIN {X 0,Y 432.825,Z 580.66,A -85,B 0,C 180,E1 8851.532,E2 8851.532} C_VEL
LIN {X 0,Y 432.736,Z 580.66,A -85,B 0,C 180,E1 8856.676,E2 8856.676} C_VEL
LIN {X 0,Y 432.705,Z 580.66,A -85,B 0,C 180,E1 8862.917,E2 8862.917} C_VEL
LIN {X 0,Y 432.811,Z 580.66,A -85,B 0,C 180,E1 8868.515,E2 8868.515} C_VEL
LIN {X 0,Y 432.903,Z 580.66,A -85,B 0,C 180,E1 8873.809,E2 8873.809} C_VEL
LIN {X 0,Y 453.139,Z 630.945,A -85,B 0,C 180,E1 8876.415,E2 8876.415} C_VEL
LIN {X 0,Y 451.262,Z 670.524,A -85,B 0,C 180,E1 8877.471,E2 8877.471} C_VEL
LIN {X 0,Y 448.234,Z 705.691,A -85,B 0,C 180,E1 8879.101,E2 8879.101} C_VEL
LIN {X 0,Y 445.4,Z 734.695,A -85,B 0,C 180,E1 8881.046,E2 8881.046} C_VEL
LIN {X 0,Y 440.165,Z 749.42,A -85,B 0,C 180,E1 8882.098,E2 8882.098} C_VEL
LIN {X 0,Y 434.768,Z 763.323,A -85,B 0,C 180,E1 8883.288,E2 8883.288} C_VEL
LIN {X 0,Y 431.603,Z 792.427,A -85,B 0,C 180,E1 8886.838,E2 8886.838} C_VEL
LIN {X 0,Y 428.95,Z 818.014,A -85,B 0,C 180,E1 8891.009,E2 8891.009} C_VEL
LIN {X 0,Y 427.52,Z 836.853,A -85,B 0,C 180,E1 8895.172,E2 8895.172} C_VEL
LIN {X 0,Y 426.82,Z 851.595,A -85,B 0,C 180,E1 8899.817,E2 8899.817} C_VEL
LIN {X 0,Y 426.624,Z 859.842,A -85,B 0,C 180,E1 8903.907,E2 8903.907} C_VEL
LIN {X 0,Y 426.573,Z 863.807,A -85,B 0,C 180,E1 8907.971,E2 8907.971} C_VEL
LIN {X 0,Y 426.715,Z 863.828,A -85,B 0,C 180,E1 8912.025,E2 8912.025} C_VEL
LIN {X 0,Y 426.597,Z 859.843,A -85,B 0,C 180,E1 8916.09,E2 8916.09} C_VEL
LIN {X 0,Y 426.863,Z 850.307,A -85,B 0,C 180,E1 8920.693,E2 8920.693} C_VEL
LIN {X 0,Y 427.776,Z 834.823,A -85,B 0,C 180,E1 8925.339,E2 8925.339} C_VEL
LIN {X 0,Y 429.433,Z 813.764,A -85,B 0,C 180,E1 8929.765,E2 8929.765} C_VEL
LIN {X 0,Y 432.218,Z 786.795,A -85,B 0,C 180,E1 8933.942,E2 8933.942} C_VEL
LIN {X 0,Y 435.517,Z 756.849,A -85,B 0,C 180,E1 8937.373,E2 8937.373} C_VEL
LIN {X 0,Y 439.138,Z 723.792,A -85,B 0,C 180,E1 8940.165,E2 8940.165} C_VEL
LIN {X 0,Y 442.875,Z 686.878,A -85,B 0,C 180,E1 8942.33,E2 8942.33} C_VEL
LIN {X 0,Y 445.708,Z 648.531,A -85,B 0,C 180,E1 8943.699,E2 8943.699} C_VEL
LIN {X 0,Y 445.704,Z 631.502,A -85,B 0,C 180,E1 8944.13,E2 8944.13} C_VEL
LIN {X 0,Y 430.301,Z 593.449,A -85,B 0,C 180,E1 8946.15,E2 8946.15} C_VEL
LIN {X 0,Y 424.886,Z 580.66,A -85,B 0,C 180,E1 8946.974,E2 8946.974} C_VEL
LIN {X 0,Y 424.782,Z 580.66,A -85,B 0,C 180,E1 8952.446,E2 8952.446} C_VEL
LIN {X 0,Y 424.886,Z 580.66,A -85,B 0,C 180,E1 8958.224,E2 8958.224} C_VEL
LIN {X 0,Y 424.862,Z 580.66,A -85,B 0,C 180,E1 8964.768,E2 8964.768} C_VEL
LIN {X 0,Y 424.943,Z 580.66,A -85,B 0,C 180,E1 8970.187,E2 8970.187} C_VEL
LIN {X 0,Y 425.244,Z 580.66,A -85,B 0,C 180,E1 8977.301,E2 8977.301} C_VEL
LIN {X 0,Y 425.339,Z 580.66,A -85,B 0,C 180,E1 8983.509,E2 8983.509} C_VEL
LIN {X 0,Y 425.499,Z 580.66,A -85,B 0,C 180,E1 8989.783,E2 8989.783} C_VEL
LIN {X 0,Y 425.821,Z 580.66,A -85,B 0,C 180,E1 8995.932,E2 8995.932} C_VEL
LIN {X 0,Y 425.921,Z 580.66,A -85,B 0,C 180,E1 9002.026,E2 9002.026} C_VEL
LIN {X 0,Y 425.664,Z 580.66,A -85,B 0,C 180,E1 9008.148,E2 9008.148} C_VEL
LIN {X 0,Y 425.493,Z 580.66,A -85,B 0,C 180,E1 9014.369,E2 9014.369} C_VEL
LIN {X 0,Y 425.264,Z 580.66,A -85,B 0,C 180,E1 9020.777,E2 9020.777} C_VEL
LIN {X 0,Y 425.028,Z 580.66,A -85,B 0,C 180,E1 9027.48,E2 9027.48} C_VEL
LIN {X 0,Y 424.925,Z 580.66,A -85,B 0,C 180,E1 9032.179,E2 9032.179} C_VEL
LIN {X 0,Y 424.791,Z 580.66,A -85,B 0,C 180,E1 9038.607,E2 9038.607} C_VEL
LIN {X 0,Y 424.853,Z 580.66,A -85,B 0,C 180,E1 9045.254,E2 9045.254} C_VEL
LIN {X 0,Y 424.894,Z 580.66,A -85,B 0,C 180,E1 9051.369,E2 9051.369} C_VEL
LIN {X 0,Y 424.926,Z 580.66,A -85,B 0,C 180,E1 9058.446,E2 9058.446} C_VEL
LIN {X 0,Y 425.012,Z 580.669,A -85,B 0,C 180,E1 9059.533,E2 9059.533} C_VEL
LIN {X 0,Y 436.277,Z 611.645,A -85,B 0,C 180,E1 9062.246,E2 9062.246} C_VEL
LIN {X 0,Y 442.143,Z 633.961,A -85,B 0,C 180,E1 9064.516,E2 9064.516} C_VEL
LIN {X 0,Y 438.5,Z 661.441,A -85,B 0,C 180,E1 9067.226,E2 9067.226} C_VEL
LIN {X 0,Y 434.88,Z 684.92,A -85,B 0,C 180,E1 9070.492,E2 9070.492} C_VEL
LIN {X 0,Y 431.593,Z 704.571,A -85,B 0,C 180,E1 9074.335,E2 9074.335} C_VEL
LIN {X 0,Y 429.441,Z 718.734,A -85,B 0,C 180,E1 9078.346,E2 9078.346} C_VEL
LIN {X 0,Y 427.934,Z 728.959,A -85,B 0,C 180,E1 9082.913,E2 9082.913} C_VEL
LIN {X 0,Y 427.596,Z 732.831,A -85,B 0,C 180,E1 9085.955,E2 9085.955} C_VEL
LIN {X 0,Y 427.27,Z 734.647,A -85,B 0,C 180,E1 9090.002,E2 9090.002} C_VEL
LIN {X 0,Y 427.725,Z 731.654,A -85,B 0,C 180,E1 9095.061,E2 9095.061} C_VEL
LIN {X 0,Y 428.789,Z 723.172,A -85,B 0,C 180,E1 9099.862,E2 9099.862} C_VEL
LIN {X 0,Y 430.815,Z 710.06,A -85,B 0,C 180,E1 9104.194,E2 9104.194} C_VEL
LIN {X 0,Y 433.739,Z 691.624,A -85,B 0,C 180,E1 9108.248,E2 9108.248} C_VEL
LIN {X 0,Y 437.539,Z 667.859,A -85,B 0,C 180,E1 9111.888,E2 9111.888} C_VEL
LIN {X 0,Y 441.281,Z 640.97,A -85,B 0,C 180,E1 9114.789,E2 9114.789} C_VEL
LIN {X 0,Y 442.03,Z 631.043,A -85,B 0,C 180,E1 9115.662,E2 9115.662} C_VEL
LIN {X 0,Y 433.092,Z 602.416,A -85,B 0,C 180,E1 9118.526,E2 9118.526} C_VEL
LIN {X 0,Y 425.009,Z 580.66,A -85,B 0,C 180,E1 9120.394,E2 9120.394} C_VEL
LIN {X 0,Y 424.882,Z 580.66,A -85,B 0,C 180,E1 9127.14,E2 9127.14} C_VEL
LIN {X 0,Y 424.85,Z 580.66,A -85,B 0,C 180,E1 9132.442,E2 9132.442} C_VEL
LIN {X 0,Y 424.868,Z 580.66,A -85,B 0,C 180,E1 9138.232,E2 9138.232} C_VEL
LIN {X 0,Y 424.84,Z 580.66,A -85,B 0,C 180,E1 9144.778,E2 9144.778} C_VEL
LIN {X 0,Y 424.899,Z 580.66,A -85,B 0,C 180,E1 9150.192,E2 9150.192} C_VEL
LIN {X 0,Y 425.202,Z 580.66,A -85,B 0,C 180,E1 9157.323,E2 9157.323} C_VEL
LIN {X 0,Y 425.307,Z 580.66,A -85,B 0,C 180,E1 9163.516,E2 9163.516} C_VEL
LIN {X 0,Y 425.491,Z 580.66,A -85,B 0,C 180,E1 9169.791,E2 9169.791} C_VEL
LIN {X 0,Y 425.843,Z 580.66,A -85,B 0,C 180,E1 9175.94,E2 9175.94} C_VEL
LIN {X 0,Y 425.86,Z 580.66,A -85,B 0,C 180,E1 9182.034,E2 9182.034} C_VEL
LIN {X 0,Y 425.691,Z 580.66,A -85,B 0,C 180,E1 9188.155,E2 9188.155} C_VEL
LIN {X 0,Y 425.499,Z 580.66,A -85,B 0,C 180,E1 9194.377,E2 9194.377} C_VEL
LIN {X 0,Y 425.261,Z 580.66,A -85,B 0,C 180,E1 9200.786,E2 9200.786} C_VEL
LIN {X 0,Y 425.042,Z 580.66,A -85,B 0,C 180,E1 9207.487,E2 9207.487} C_VEL
LIN {X 0,Y 424.904,Z 580.66,A -85,B 0,C 180,E1 9212.19,E2 9212.19} C_VEL
LIN {X 0,Y 424.772,Z 580.66,A -85,B 0,C 180,E1 9218.599,E2 9218.599} C_VEL
LIN {X 0,Y 424.859,Z 580.66,A -85,B 0,C 180,E1 9225.264,E2 9225.264} C_VEL
LIN {X 0,Y 424.905,Z 580.66,A -85,B 0,C 180,E1 9231.38,E2 9231.38} C_VEL
LIN {X 0,Y 424.968,Z 580.66,A -85,B 0,C 180,E1 9233.087,E2 9233.087} C_VEL
LIN {X 0,Y 443.679,Z 626.076,A -85,B 0,C 180,E1 9235.61,E2 9235.61} C_VEL
LIN {X 0,Y 446.309,Z 634.535,A -85,B 0,C 180,E1 9235.988,E2 9235.988} C_VEL
LIN {X 0,Y 444.117,Z 672.478,A -85,B 0,C 180,E1 9237.068,E2 9237.068} C_VEL
LIN {X 0,Y 440.739,Z 709.097,A -85,B 0,C 180,E1 9238.863,E2 9238.863} C_VEL
LIN {X 0,Y 436.976,Z 744.204,A -85,B 0,C 180,E1 9241.455,E2 9241.455} C_VEL
LIN {X 0,Y 434.768,Z 763.323,A -85,B 0,C 180,E1 9243.288,E2 9243.288} C_VEL
LIN {X 0,Y 429.296,Z 776.688,A -85,B 0,C 180,E1 9244.637,E2 9244.637} C_VEL
LIN {X 0,Y 424.197,Z 789.075,A -85,B 0,C 180,E1 9246.136,E2 9246.136} C_VEL
LIN {X 0,Y 421.397,Z 815.169,A -85,B 0,C 180,E1 9250.383,E2 9250.383} C_VEL
LIN {X 0,Y 419.714,Z 835.448,A -85,B 0,C 180,E1 9254.89,E2 9254.89} C_VEL
LIN {X 0,Y 418.983,Z 850.278,A -85,B 0,C 180,E1 9259.624,E2 9259.624} C_VEL
LIN {X 0,Y 418.794,Z 858.609,A -85,B 0,C 180,E1 9263.793,E2 9263.793} C_VEL
LIN {X 0,Y 418.772,Z 862.617,A -85,B 0,C 180,E1 9267.933,E2 9267.933} C_VEL
LIN {X 0,Y 418.9,Z 862.636,A -85,B 0,C 180,E1 9272.063,E2 9272.063} C_VEL
LIN {X 0,Y 418.838,Z 857.26,A -85,B 0,C 180,E1 9277.028,E2 9277.028} C_VEL
LIN {X 0,Y 419.084,Z 847.498,A -85,B 0,C 180,E1 9281.42,E2 9281.42} C_VEL
LIN {X 0,Y 420.06,Z 831.25,A -85,B 0,C 180,E1 9286.162,E2 9286.162} C_VEL
LIN {X 0,Y 421.945,Z 809.418,A -85,B 0,C 180,E1 9290.678,E2 9290.678} C_VEL
LIN {X 0,Y 424.989,Z 782.204,A -85,B 0,C 180,E1 9294.795,E2 9294.795} C_VEL
LIN {X 0,Y 428.762,Z 751.266,A -85,B 0,C 180,E1 9298.271,E2 9298.271} C_VEL
LIN {X 0,Y 432.694,Z 716.548,A -85,B 0,C 180,E1 9301.099,E2 9301.099} C_VEL
LIN {X 0,Y 436.432,Z 679.586,A -85,B 0,C 180,E1 9303.139,E2 9303.139} C_VEL
LIN {X 0,Y 439.257,Z 640.444,A -85,B 0,C 180,E1 9304.416,E2 9304.416} C_VEL
LIN {X 0,Y 438.535,Z 632.76,A -85,B 0,C 180,E1 9304.654,E2 9304.654} C_VEL
LIN {X 0,Y 424.006,Z 596.842,A -85,B 0,C 180,E1 9306.627,E2 9306.627} C_VEL
LIN {X 0,Y 416.939,Z 580.66,A -85,B 0,C 180,E1 9307.641,E2 9307.641} C_VEL
LIN {X 0,Y 416.822,Z 580.66,A -85,B 0,C 180,E1 9313.61,E2 9313.61} C_VEL
LIN {X 0,Y 416.919,Z 580.66,A -85,B 0,C 180,E1 9319.464,E2 9319.464} C_VEL
LIN {X 0,Y 416.949,Z 580.66,A -85,B 0,C 180,E1 9324.614,E2 9324.614} C_VEL
LIN {X 0,Y 417.043,Z 580.66,A -85,B 0,C 180,E1 9331.939,E2 9331.939} C_VEL
LIN {X 0,Y 417.339,Z 580.66,A -85,B 0,C 180,E1 9338.801,E2 9338.801} C_VEL
LIN {X 0,Y 417.431,Z 580.66,A -85,B 0,C 180,E1 9345.339,E2 9345.339} C_VEL
LIN {X 0,Y 417.718,Z 580.66,A -85,B 0,C 180,E1 9351.689,E2 9351.689} C_VEL
LIN {X 0,Y 418.148,Z 580.66,A -85,B 0,C 180,E1 9357.928,E2 9357.928} C_VEL
LIN {X 0,Y 418.065,Z 580.66,A -85,B 0,C 180,E1 9364.135,E2 9364.135} C_VEL
LIN {X 0,Y 417.681,Z 580.66,A -85,B 0,C 180,E1 9370.402,E2 9370.402} C_VEL
LIN {X 0,Y 417.485,Z 580.66,A -85,B 0,C 180,E1 9376.802,E2 9376.802} C_VEL
LIN {X 0,Y 417.267,Z 580.66,A -85,B 0,C 180,E1 9383.434,E2 9383.434} C_VEL
LIN {X 0,Y 417.024,Z 580.66,A -85,B 0,C 180,E1 9390.429,E2 9390.429} C_VEL
LIN {X 0,Y 416.898,Z 580.66,A -85,B 0,C 180,E1 9397.967,E2 9397.967} C_VEL
LIN {X 0,Y 416.845,Z 580.66,A -85,B 0,C 180,E1 9403.619,E2 9403.619} C_VEL
LIN {X 0,Y 416.953,Z 580.66,A -85,B 0,C 180,E1 9409.453,E2 9409.453} C_VEL
LIN {X 0,Y 416.932,Z 580.66,A -85,B 0,C 180,E1 9414.618,E2 9414.618} C_VEL
LIN {X 0,Y 417.071,Z 580.814,A -85,B 0,C 180,E1 9418.791,E2 9418.791} C_VEL
LIN {X 0,Y 428.699,Z 612.191,A -85,B 0,C 180,E1 9421.623,E2 9421.623} C_VEL
LIN {X 0,Y 435.154,Z 635.487,A -85,B 0,C 180,E1 9424.083,E2 9424.083} C_VEL
LIN {X 0,Y 431.344,Z 662.8,A -85,B 0,C 180,E1 9426.827,E2 9426.827} C_VEL
LIN {X 0,Y 427.526,Z 686.202,A -85,B 0,C 180,E1 9430.143,E2 9430.143} C_VEL
LIN {X 0,Y 424.026,Z 706.062,A -85,B 0,C 180,E1 9434.106,E2 9434.106} C_VEL
LIN {X 0,Y 421.518,Z 721.346,A -85,B 0,C 180,E1 9438.647,E2 9438.647} C_VEL
LIN {X 0,Y 420.18,Z 730.156,A -85,B 0,C 180,E1 9442.781,E2 9442.781} C_VEL
LIN {X 0,Y 419.817,Z 734.018,A -85,B 0,C 180,E1 9445.88,E2 9445.88} C_VEL
LIN {X 0,Y 419.484,Z 735.83,A -85,B 0,C 180,E1 9450.002,E2 9450.002} C_VEL
LIN {X 0,Y 419.967,Z 732.842,A -85,B 0,C 180,E1 9455.155,E2 9455.155} C_VEL
LIN {X 0,Y 420.962,Z 725.354,A -85,B 0,C 180,E1 9459.629,E2 9459.629} C_VEL
LIN {X 0,Y 422.943,Z 713.09,A -85,B 0,C 180,E1 9463.937,E2 9463.937} C_VEL
LIN {X 0,Y 425.914,Z 695.606,A -85,B 0,C 180,E1 9468.061,E2 9468.061} C_VEL
LIN {X 0,Y 429.713,Z 673.097,A -85,B 0,C 180,E1 9471.751,E2 9471.751} C_VEL
LIN {X 0,Y 433.679,Z 646.663,A -85,B 0,C 180,E1 9474.814,E2 9474.814} C_VEL
LIN {X 0,Y 434.79,Z 632.825,A -85,B 0,C 180,E1 9476.103,E2 9476.103} C_VEL
LIN {X 0,Y 425.755,Z 603.567,A -85,B 0,C 180,E1 9479.11,E2 9479.11} C_VEL
LIN {X 0,Y 417.034,Z 580.66,A -85,B 0,C 180,E1 9481.12,E2 9481.12} C_VEL
LIN {X 0,Y 416.954,Z 580.66,A -85,B 0,C 180,E1 9487.97,E2 9487.97} C_VEL
LIN {X 0,Y 416.866,Z 580.66,A -85,B 0,C 180,E1 9493.628,E2 9493.628} C_VEL
LIN {X 0,Y 416.908,Z 580.66,A -85,B 0,C 180,E1 9499.471,E2 9499.471} C_VEL
LIN {X 0,Y 416.926,Z 580.66,A -85,B 0,C 180,E1 9504.622,E2 9504.622} C_VEL
LIN {X 0,Y 417.018,Z 580.66,A -85,B 0,C 180,E1 9511.946,E2 9511.946} C_VEL
LIN {X 0,Y 417.324,Z 580.66,A -85,B 0,C 180,E1 9518.808,E2 9518.808} C_VEL
LIN {X 0,Y 417.376,Z 580.66,A -85,B 0,C 180,E1 9525.346,E2 9525.346} C_VEL
LIN {X 0,Y 417.728,Z 580.66,A -85,B 0,C 180,E1 9531.697,E2 9531.697} C_VEL
LIN {X 0,Y 418.174,Z 580.66,A -85,B 0,C 180,E1 9537.936,E2 9537.936} C_VEL
LIN {X 0,Y 417.955,Z 580.66,A -85,B 0,C 180,E1 9544.144,E2 9544.144} C_VEL
LIN {X 0,Y 417.713,Z 580.66,A -85,B 0,C 180,E1 9550.409,E2 9550.409} C_VEL
LIN {X 0,Y 417.478,Z 580.66,A -85,B 0,C 180,E1 9556.81,E2 9556.81} C_VEL
LIN {X 0,Y 417.218,Z 580.66,A -85,B 0,C 180,E1 9563.446,E2 9563.446} C_VEL
LIN {X 0,Y 417.021,Z 580.66,A -85,B 0,C 180,E1 9570.439,E2 9570.439} C_VEL
LIN {X 0,Y 416.859,Z 580.66,A -85,B 0,C 180,E1 9577.981,E2 9577.981} C_VEL
LIN {X 0,Y 416.836,Z 580.66,A -85,B 0,C 180,E1 9583.613,E2 9583.613} C_VEL
LIN {X 0,Y 416.936,Z 580.66,A -85,B 0,C 180,E1 9589.468,E2 9589.468} C_VEL
LIN {X 0,Y 417.029,Z 581.166,A -85,B 0,C 180,E1 9592.404,E2 9592.404} C_VEL
LIN {X 0,Y 435.885,Z 625.332,A -85,B 0,C 180,E1 9594.98,E2 9594.98} C_VEL
LIN {X 0,Y 439.455,Z 635.954,A -85,B 0,C 180,E1 9595.497,E2 9595.497} C_VEL
LIN {X 0,Y 436.917,Z 675.16,A -85,B 0,C 180,E1 9596.677,E2 9596.677} C_VEL
LIN {X 0,Y 433.204,Z 712.548,A -85,B 0,C 180,E1 9598.646,E2 9598.646} C_VEL
LIN {X 0,Y 429.266,Z 746.86,A -85,B 0,C 180,E1 9601.316,E2 9601.316} C_VEL
LIN {X 0,Y 425.351,Z 779.093,A -85,B 0,C 180,E1 9604.803,E2 9604.803} C_VEL
LIN {X 0,Y 424.197,Z 789.075,A -85,B 0,C 180,E1 9606.136,E2 9606.136} C_VEL
LIN {X 0,Y 422.352,Z 795.1,A -85,B 0,C 180,E1 9606.971,E2 9606.971} C_VEL
LIN {X 0,Y 414.162,Z 810.142,A -85,B 0,C 180,E1 9609.32,E2 9609.32} C_VEL
LIN {X 0,Y 413.967,Z 811.424,A -85,B 0,C 180,E1 9609.562,E2 9609.562} C_VEL
LIN {X 0,Y 412.011,Z 833.087,A -85,B 0,C 180,E1 9614.328,E2 9614.328} C_VEL
LIN {X 0,Y 411.177,Z 847.667,A -85,B 0,C 180,E1 9618.89,E2 9618.89} C_VEL
LIN {X 0,Y 410.978,Z 857.379,A -85,B 0,C 180,E1 9623.674,E2 9623.674} C_VEL
LIN {X 0,Y 410.952,Z 861.422,A -85,B 0,C 180,E1 9627.894,E2 9627.894} C_VEL
LIN {X 0,Y 411.076,Z 861.442,A -85,B 0,C 180,E1 9632.102,E2 9632.102} C_VEL
LIN {X 0,Y 410.954,Z 857.381,A -85,B 0,C 180,E1 9636.322,E2 9636.322} C_VEL
LIN {X 0,Y 411.192,Z 847.674,A -85,B 0,C 180,E1 9641.106,E2 9641.106} C_VEL
LIN {X 0,Y 412.119,Z 832.038,A -85,B 0,C 180,E1 9645.936,E2 9645.936} C_VEL
LIN {X 0,Y 413.993,Z 810.91,A -85,B 0,C 180,E1 9650.535,E2 9650.535} C_VEL
LIN {X 0,Y 417.193,Z 783.298,A -85,B 0,C 180,E1 9654.931,E2 9654.931} C_VEL
LIN {X 0,Y 421.097,Z 752.981,A -85,B 0,C 180,E1 9658.474,E2 9658.474} C_VEL
LIN {X 0,Y 425.376,Z 717.923,A -85,B 0,C 180,E1 9661.458,E2 9661.458} C_VEL
LIN {X 0,Y 429.398,Z 680.392,A -85,B 0,C 180,E1 9663.603,E2 9663.603} C_VEL
LIN {X 0,Y 432.385,Z 643.061,A -85,B 0,C 180,E1 9664.883,E2 9664.883} C_VEL
LIN {X 0,Y 431.709,Z 634.772,A -85,B 0,C 180,E1 9665.153,E2 9665.153} C_VEL
LIN {X 0,Y 417.291,Z 599.091,A -85,B 0,C 180,E1 9667.185,E2 9667.185} C_VEL
LIN {X 0,Y 408.955,Z 580.66,A -85,B 0,C 180,E1 9668.416,E2 9668.416} C_VEL
LIN {X 0,Y 408.861,Z 580.66,A -85,B 0,C 180,E1 9675.473,E2 9675.473} C_VEL
LIN {X 0,Y 408.964,Z 580.66,A -85,B 0,C 180,E1 9681.15,E2 9681.15} C_VEL
LIN {X 0,Y 408.993,Z 580.66,A -85,B 0,C 180,E1 9688.051,E2 9688.051} C_VEL
LIN {X 0,Y 409.174,Z 580.66,A -85,B 0,C 180,E1 9693.731,E2 9693.731} C_VEL
LIN {X 0,Y 409.452,Z 580.66,A -85,B 0,C 180,E1 9700.626,E2 9700.626} C_VEL
LIN {X 0,Y 409.605,Z 580.66,A -85,B 0,C 180,E1 9707.227,E2 9707.227} C_VEL
LIN {X 0,Y 409.978,Z 580.66,A -85,B 0,C 180,E1 9713.657,E2 9713.657} C_VEL
LIN {X 0,Y 410.178,Z 580.66,A -85,B 0,C 180,E1 9719.996,E2 9719.996} C_VEL
LIN {X 0,Y 409.964,Z 580.66,A -85,B 0,C 180,E1 9726.418,E2 9726.418} C_VEL
LIN {X 0,Y 409.723,Z 580.66,A -85,B 0,C 180,E1 9732.761,E2 9732.761} C_VEL
LIN {X 0,Y 409.453,Z 580.66,A -85,B 0,C 180,E1 9739.365,E2 9739.365} C_VEL
LIN {X 0,Y 409.179,Z 580.66,A -85,B 0,C 180,E1 9746.259,E2 9746.259} C_VEL
LIN {X 0,Y 408.999,Z 580.66,A -85,B 0,C 180,E1 9753.594,E2 9753.594} C_VEL
LIN {X 0,Y 408.866,Z 580.66,A -85,B 0,C 180,E1 9759.198,E2 9759.198} C_VEL
LIN {X 0,Y 408.872,Z 580.66,A -85,B 0,C 180,E1 9765.481,E2 9765.481} C_VEL
LIN {X 0,Y 408.975,Z 580.66,A -85,B 0,C 180,E1 9771.157,E2 9771.157} C_VEL
LIN {X 0,Y 409.114,Z 581.076,A -85,B 0,C 180,E1 9778.016,E2 9778.016} C_VEL
LIN {X 0,Y 421.028,Z 612.219,A -85,B 0,C 180,E1 9780.928,E2 9780.928} C_VEL
LIN {X 0,Y 427.944,Z 638.552,A -85,B 0,C 180,E1 9783.766,E2 9783.766} C_VEL
LIN {X 0,Y 423.85,Z 666.244,A -85,B 0,C 180,E1 9786.67,E2 9786.67} C_VEL
LIN {X 0,Y 419.677,Z 690.466,A -85,B 0,C 180,E1 9790.303,E2 9790.303} C_VEL
LIN {X 0,Y 416.003,Z 710.144,A -85,B 0,C 180,E1 9794.544,E2 9794.544} C_VEL
LIN {X 0,Y 413.649,Z 723.947,A -85,B 0,C 180,E1 9798.961,E2 9798.961} C_VEL
LIN {X 0,Y 412.371,Z 732.844,A -85,B 0,C 180,E1 9803.7,E2 9803.7} C_VEL
LIN {X 0,Y 411.944,Z 736.504,A -85,B 0,C 180,E1 9807.903,E2 9807.903} C_VEL
LIN {X 0,Y 411.952,Z 736.459,A -85,B 0,C 180,E1 9812.101,E2 9812.101} C_VEL
LIN {X 0,Y 412.453,Z 732.701,A -85,B 0,C 180,E1 9816.303,E2 9816.303} C_VEL
LIN {X 0,Y 413.661,Z 723.694,A -85,B 0,C 180,E1 9821.042,E2 9821.042} C_VEL
LIN {X 0,Y 416.138,Z 709.639,A -85,B 0,C 180,E1 9825.488,E2 9825.488} C_VEL
LIN {X 0,Y 419.741,Z 689.917,A -85,B 0,C 180,E1 9829.697,E2 9829.697} C_VEL
LIN {X 0,Y 423.956,Z 665.512,A -85,B 0,C 180,E1 9833.327,E2 9833.327} C_VEL
LIN {X 0,Y 428.001,Z 638.307,A -85,B 0,C 180,E1 9836.154,E2 9836.154} C_VEL
LIN {X 0,Y 420.941,Z 612.158,A -85,B 0,C 180,E1 9838.984,E2 9838.984} C_VEL
LIN {X 0,Y 409.095,Z 580.66,A -85,B 0,C 180,E1 9841.98,E2 9841.98} C_VEL
LIN {X 0,Y 408.939,Z 580.66,A -85,B 0,C 180,E1 9848.851,E2 9848.851} C_VEL
LIN {X 0,Y 408.874,Z 580.66,A -85,B 0,C 180,E1 9855.486,E2 9855.486} C_VEL
LIN {X 0,Y 408.949,Z 580.66,A -85,B 0,C 180,E1 9861.159,E2 9861.159} C_VEL
LIN {X 0,Y 408.989,Z 580.66,A -85,B 0,C 180,E1 9866.405,E2 9866.405} C_VEL
LIN {X 0,Y 409.131,Z 580.66,A -85,B 0,C 180,E1 9873.737,E2 9873.737} C_VEL
LIN {X 0,Y 409.453,Z 580.66,A -85,B 0,C 180,E1 9880.635,E2 9880.635} C_VEL
LIN {X 0,Y 409.535,Z 580.66,A -85,B 0,C 180,E1 9887.233,E2 9887.233} C_VEL
LIN {X 0,Y 409.997,Z 580.66,A -85,B 0,C 180,E1 9893.665,E2 9893.665} C_VEL
LIN {X 0,Y 410.192,Z 580.66,A -85,B 0,C 180,E1 9900.004,E2 9900.004} C_VEL
LIN {X 0,Y 409.949,Z 580.66,A -85,B 0,C 180,E1 9906.367,E2 9906.367} C_VEL
LIN {X 0,Y 409.751,Z 580.66,A -85,B 0,C 180,E1 9912.768,E2 9912.768} C_VEL
LIN {X 0,Y 409.445,Z 580.66,A -85,B 0,C 180,E1 9919.374,E2 9919.374} C_VEL
LIN {X 0,Y 409.159,Z 580.66,A -85,B 0,C 180,E1 9926.269,E2 9926.269} C_VEL
LIN {X 0,Y 408.992,Z 580.66,A -85,B 0,C 180,E1 9933.604,E2 9933.604} C_VEL
LIN {X 0,Y 408.845,Z 580.66,A -85,B 0,C 180,E1 9939.188,E2 9939.188} C_VEL
LIN {X 0,Y 408.875,Z 580.66,A -85,B 0,C 180,E1 9945.476,E2 9945.476} C_VEL
LIN {X 0,Y 409.04,Z 580.66,A -85,B 0,C 180,E1 9951.59,E2 9951.59} C_VEL
LIN {X 0,Y 428.886,Z 626.715,A -85,B 0,C 180,E1 9954.432,E2 9954.432} C_VEL
LIN {X 0,Y 432.62,Z 638.679,A -85,B 0,C 180,E1 9955.02,E2 9955.02} C_VEL
LIN {X 0,Y 429.736,Z 677.431,A -85,B 0,C 180,E1 9956.272,E2 9956.272} C_VEL
LIN {X 0,Y 425.857,Z 714.08,A -85,B 0,C 180,E1 9958.292,E2 9958.292} C_VEL
LIN {X 0,Y 421.687,Z 748.334,A -85,B 0,C 180,E1 9961.063,E2 9961.063} C_VEL
LIN {X 0,Y 417.664,Z 779.605,A -85,B 0,C 180,E1 9964.585,E2 9964.585} C_VEL
LIN {X 0,Y 414.467,Z 806.419,A -85,B 0,C 180,E1 9968.648,E2 9968.648} C_VEL
LIN {X 0,Y 413.967,Z 811.424,A -85,B 0,C 180,E1 9969.562,E2 9969.562} C_VEL
LIN {X 0,Y 412.293,Z 816.506,A -85,B 0,C 180,E1 9970.528,E2 9970.528} C_VEL
LIN {X 0,Y 404.526,Z 828.809,A -85,B 0,C 180,E1 9973.256,E2 9973.256} C_VEL
LIN {X 0,Y 404.36,Z 829.855,A -85,B 0,C 180,E1 9973.527,E2 9973.527} C_VEL
LIN {X 0,Y 403.415,Z 844.915,A -85,B 0,C 180,E1 9978.127,E2 9978.127} C_VEL
LIN {X 0,Y 403.165,Z 855.119,A -85,B 0,C 180,E1 9982.9,E2 9982.9} C_VEL
LIN {X 0,Y 403.131,Z 860.229,A -85,B 0,C 180,E1 9987.853,E2 9987.853} C_VEL
LIN {X 0,Y 403.275,Z 860.253,A -85,B 0,C 180,E1 9992.143,E2 9992.143} C_VEL
LIN {X 0,Y 403.149,Z 855.13,A -85,B 0,C 180,E1 9997.091,E2 9997.091} C_VEL
LIN {X 0,Y 403.399,Z 844.917,A -85,B 0,C 180,E1 10001.87,E2 10001.87} C_VEL
LIN {X 0,Y 404.317,Z 829.629,A -85,B 0,C 180,E1 10006.531,E2 10006.531} C_VEL
LIN {X 0,Y 406.44,Z 808.086,A -85,B 0,C 180,E1 10011.219,E2 10011.219} C_VEL
LIN {X 0,Y 409.831,Z 780.953,A -85,B 0,C 180,E1 10015.537,E2 10015.537} C_VEL
LIN {X 0,Y 414.007,Z 750.417,A -85,B 0,C 180,E1 10019.123,E2 10019.123} C_VEL
LIN {X 0,Y 418.521,Z 715.722,A -85,B 0,C 180,E1 10022.073,E2 10022.073} C_VEL
LIN {X 0,Y 422.56,Z 679.819,A -85,B 0,C 180,E1 10024.144,E2 10024.144} C_VEL
LIN {X 0,Y 425.747,Z 640.724,A -85,B 0,C 180,E1 10025.497,E2 10025.497} C_VEL
LIN {X 0,Y 415.792,Z 612.905,A -85,B 0,C 180,E1 10027.02,E2 10027.02} C_VEL
LIN {X 0,Y 400.99,Z 580.66,A -85,B 0,C 180,E1 10029.23,E2 10029.23} C_VEL
LIN {X 0,Y 400.954,Z 580.66,A -85,B 0,C 180,E1 10035.643,E2 10035.643} C_VEL
LIN {X 0,Y 401.015,Z 580.66,A -85,B 0,C 180,E1 10042.981,E2 10042.981} C_VEL
LIN {X 0,Y 401.08,Z 580.66,A -85,B 0,C 180,E1 10049.912,E2 10049.912} C_VEL
LIN {X 0,Y 401.302,Z 580.66,A -85,B 0,C 180,E1 10055.565,E2 10055.565} C_VEL
LIN {X 0,Y 401.551,Z 580.66,A -85,B 0,C 180,E1 10062.502,E2 10062.502} C_VEL
LIN {X 0,Y 401.732,Z 580.66,A -85,B 0,C 180,E1 10069.172,E2 10069.172} C_VEL
LIN {X 0,Y 402.108,Z 580.66,A -85,B 0,C 180,E1 10075.692,E2 10075.692} C_VEL
LIN {X 0,Y 402.247,Z 580.66,A -85,B 0,C 180,E1 10082.146,E2 10082.146} C_VEL
LIN {X 0,Y 401.891,Z 580.66,A -85,B 0,C 180,E1 10088.633,E2 10088.633} C_VEL
LIN {X 0,Y 401.703,Z 580.66,A -85,B 0,C 180,E1 10095.24,E2 10095.24} C_VEL
LIN {X 0,Y 401.436,Z 580.66,A -85,B 0,C 180,E1 10102.073,E2 10102.073} C_VEL
LIN {X 0,Y 401.127,Z 580.66,A -85,B 0,C 180,E1 10109.27,E2 10109.27} C_VEL
LIN {X 0,Y 401.052,Z 580.66,A -85,B 0,C 180,E1 10114.351,E2 10114.351} C_VEL
LIN {X 0,Y 400.894,Z 580.66,A -85,B 0,C 180,E1 10121.171,E2 10121.171} C_VEL
LIN {X 0,Y 400.981,Z 580.66,A -85,B 0,C 180,E1 10127.366,E2 10127.366} C_VEL
LIN {X 0,Y 401.007,Z 580.66,A -85,B 0,C 180,E1 10132.985,E2 10132.985} C_VEL
LIN {X 0,Y 401.128,Z 580.782,A -85,B 0,C 180,E1 10137.178,E2 10137.178} C_VEL
LIN {X 0,Y 413.448,Z 612.627,A -85,B 0,C 180,E1 10140.238,E2 10140.238} C_VEL
LIN {X 0,Y 421.037,Z 639.733,A -85,B 0,C 180,E1 10143.277,E2 10143.277} C_VEL
LIN {X 0,Y 416.721,Z 667.563,A -85,B 0,C 180,E1 10146.247,E2 10146.247} C_VEL
LIN {X 0,Y 412.331,Z 691.738,A -85,B 0,C 180,E1 10149.937,E2 10149.937} C_VEL
LIN {X 0,Y 408.673,Z 710.21,A -85,B 0,C 180,E1 10153.938,E2 10153.938} C_VEL
LIN {X 0,Y 405.964,Z 725.156,A -85,B 0,C 180,E1 10158.749,E2 10158.749} C_VEL
LIN {X 0,Y 404.587,Z 734.039,A -85,B 0,C 180,E1 10163.578,E2 10163.578} C_VEL
LIN {X 0,Y 404.162,Z 737.687,A -85,B 0,C 180,E1 10167.862,E2 10167.862} C_VEL
LIN {X 0,Y 404.17,Z 737.643,A -85,B 0,C 180,E1 10172.141,E2 10172.141} C_VEL
LIN {X 0,Y 404.672,Z 733.896,A -85,B 0,C 180,E1 10176.424,E2 10176.424} C_VEL
LIN {X 0,Y 406.004,Z 724.904,A -85,B 0,C 180,E1 10181.253,E2 10181.253} C_VEL
LIN {X 0,Y 408.804,Z 709.605,A -85,B 0,C 180,E1 10186.124,E2 10186.124} C_VEL
LIN {X 0,Y 412.703,Z 689.693,A -85,B 0,C 180,E1 10190.326,E2 10190.326} C_VEL
LIN {X 0,Y 416.993,Z 665.803,A -85,B 0,C 180,E1 10193.882,E2 10193.882} C_VEL
LIN {X 0,Y 420.795,Z 638.365,A -85,B 0,C 180,E1 10196.782,E2 10196.782} C_VEL
LIN {X 0,Y 412.318,Z 609.198,A -85,B 0,C 180,E1 10200.013,E2 10200.013} C_VEL
LIN {X 0,Y 401.106,Z 580.66,A -85,B 0,C 180,E1 10202.764,E2 10202.764} C_VEL
LIN {X 0,Y 400.971,Z 580.66,A -85,B 0,C 180,E1 10209.774,E2 10209.774} C_VEL
LIN {X 0,Y 400.963,Z 580.66,A -85,B 0,C 180,E1 10215.647,E2 10215.647} C_VEL
LIN {X 0,Y 400.997,Z 580.66,A -85,B 0,C 180,E1 10222.989,E2 10222.989} C_VEL
LIN {X 0,Y 401.05,Z 580.66,A -85,B 0,C 180,E1 10229.927,E2 10229.927} C_VEL
LIN {X 0,Y 401.268,Z 580.66,A -85,B 0,C 180,E1 10235.572,E2 10235.572} C_VEL
LIN {X 0,Y 401.538,Z 580.66,A -85,B 0,C 180,E1 10242.51,E2 10242.51} C_VEL
LIN {X 0,Y 401.709,Z 580.66,A -85,B 0,C 180,E1 10249.179,E2 10249.179} C_VEL
LIN {X 0,Y 402.129,Z 580.66,A -85,B 0,C 180,E1 10255.7,E2 10255.7} C_VEL
LIN {X 0,Y 402.306,Z 580.66,A -85,B 0,C 180,E1 10260.004,E2 10260.004} C_VEL
LIN {X 0,Y 402.058,Z 580.66,A -85,B 0,C 180,E1 10266.468,E2 10266.468} C_VEL
LIN {X 0,Y 401.825,Z 580.66,A -85,B 0,C 180,E1 10273.025,E2 10273.025} C_VEL
LIN {X 0,Y 401.459,Z 580.66,A -85,B 0,C 180,E1 10280.003,E2 10280.003} C_VEL
LIN {X 0,Y 401.227,Z 580.66,A -85,B 0,C 180,E1 10286.83,E2 10286.83} C_VEL
LIN {X 0,Y 401.026,Z 580.66,A -85,B 0,C 180,E1 10294.364,E2 10294.364} C_VEL
LIN {X 0,Y 400.88,Z 580.66,A -85,B 0,C 180,E1 10301.164,E2 10301.164} C_VEL
LIN {X 0,Y 400.984,Z 580.66,A -85,B 0,C 180,E1 10307.361,E2 10307.361} C_VEL
LIN {X 0,Y 401.092,Z 580.902,A -85,B 0,C 180,E1 10310.832,E2 10310.832} C_VEL
LIN {X 0,Y 422.05,Z 628.361,A -85,B 0,C 180,E1 10313.883,E2 10313.883} C_VEL
LIN {X 0,Y 425.82,Z 640.585,A -85,B 0,C 180,E1 10314.511,E2 10314.511} C_VEL
LIN {X 0,Y 422.612,Z 679.663,A -85,B 0,C 180,E1 10315.857,E2 10315.857} C_VEL
LIN {X 0,Y 418.549,Z 715.627,A -85,B 0,C 180,E1 10317.926,E2 10317.926} C_VEL
LIN {X 0,Y 414.104,Z 749.735,A -85,B 0,C 180,E1 10320.811,E2 10320.811} C_VEL
LIN {X 0,Y 409.856,Z 780.933,A -85,B 0,C 180,E1 10324.463,E2 10324.463} C_VEL
LIN {X 0,Y 406.482,Z 808.069,A -85,B 0,C 180,E1 10328.779,E2 10328.779} C_VEL
LIN {X 0,Y 404.36,Z 829.855,A -85,B 0,C 180,E1 10333.527,E2 10333.527} C_VEL
LIN {X 0,Y 402.844,Z 833.897,A -85,B 0,C 180,E1 10334.612,E2 10334.612} C_VEL
LIN {X 0,Y 395.675,Z 843.091,A -85,B 0,C 180,E1 10337.675,E2 10337.675} C_VEL
LIN {X 0,Y 395.544,Z 843.873,A -85,B 0,C 180,E1 10337.972,E2 10337.972} C_VEL
LIN {X 0,Y 395.35,Z 854.152,A -85,B 0,C 180,E1 10342.916,E2 10342.916} C_VEL
LIN {X 0,Y 395.309,Z 859.038,A -85,B 0,C 180,E1 10347.811,E2 10347.811} C_VEL
LIN {X 0,Y 395.448,Z 859.061,A -85,B 0,C 180,E1 10352.185,E2 10352.185} C_VEL
LIN {X 0,Y 395.332,Z 854.183,A -85,B 0,C 180,E1 10357.063,E2 10357.063} C_VEL
LIN {X 0,Y 395.536,Z 843.65,A -85,B 0,C 180,E1 10362.11,E2 10362.11} C_VEL
LIN {X 0,Y 396.633,Z 827.248,A -85,B 0,C 180,E1 10367.146,E2 10367.146} C_VEL
LIN {X 0,Y 399.002,Z 805.244,A -85,B 0,C 180,E1 10371.926,E2 10371.926} C_VEL
LIN {X 0,Y 402.66,Z 778.008,A -85,B 0,C 180,E1 10376.248,E2 10376.248} C_VEL
LIN {X 0,Y 407.115,Z 746.943,A -85,B 0,C 180,E1 10379.891,E2 10379.891} C_VEL
LIN {X 0,Y 411.852,Z 712.78,A -85,B 0,C 180,E1 10382.758,E2 10382.758} C_VEL
LIN {X 0,Y 415.951,Z 677.87,A -85,B 0,C 180,E1 10384.763,E2 10384.763} C_VEL
LIN {X 0,Y 418.594,Z 640.081,A -85,B 0,C 180,E1 10386.124,E2 10386.124} C_VEL
LIN {X 0,Y 405.016,Z 606.265,A -85,B 0,C 180,E1 10388.196,E2 10388.196} C_VEL
LIN {X 0,Y 393.026,Z 580.66,A -85,B 0,C 180,E1 10390.086,E2 10390.086} C_VEL
LIN {X 0,Y 393.045,Z 580.66,A -85,B 0,C 180,E1 10396.835,E2 10396.835} C_VEL
LIN {X 0,Y 393.067,Z 580.66,A -85,B 0,C 180,E1 10403.719,E2 10403.719} C_VEL
LIN {X 0,Y 393.194,Z 580.66,A -85,B 0,C 180,E1 10410.07,E2 10410.07} C_VEL
LIN {X 0,Y 393.443,Z 580.66,A -85,B 0,C 180,E1 10417.445,E2 10417.445} C_VEL
LIN {X 0,Y 393.654,Z 580.66,A -85,B 0,C 180,E1 10424.432,E2 10424.432} C_VEL
LIN {X 0,Y 393.934,Z 580.66,A -85,B 0,C 180,E1 10431.183,E2 10431.183} C_VEL
LIN {X 0,Y 394.435,Z 580.66,A -85,B 0,C 180,E1 10437.804,E2 10437.804} C_VEL
LIN {X 0,Y 394.321,Z 580.66,A -85,B 0,C 180,E1 10444.385,E2 10444.385} C_VEL
LIN {X 0,Y 393.914,Z 580.66,A -85,B 0,C 180,E1 10451.037,E2 10451.037} C_VEL
LIN {X 0,Y 393.63,Z 580.66,A -85,B 0,C 180,E1 10457.853,E2 10457.853} C_VEL
LIN {X 0,Y 393.377,Z 580.66,A -85,B 0,C 180,E1 10464.951,E2 10464.951} C_VEL
LIN {X 0,Y 393.118,Z 580.66,A -85,B 0,C 180,E1 10472.498,E2 10472.498} C_VEL
LIN {X 0,Y 393.033,Z 580.66,A -85,B 0,C 180,E1 10479.843,E2 10479.843} C_VEL
LIN {X 0,Y 393.049,Z 580.66,A -85,B 0,C 180,E1 10486.829,E2 10486.829} C_VEL
LIN {X 0,Y 393.054,Z 580.66,A -85,B 0,C 180,E1 10493.715,E2 10493.715} C_VEL
LIN {X 0,Y 393.215,Z 581.352,A -85,B 0,C 180,E1 10496.341,E2 10496.341} C_VEL
LIN {X 0,Y 405.891,Z 612.857,A -85,B 0,C 180,E1 10499.506,E2 10499.506} C_VEL
LIN {X 0,Y 413.801,Z 641.089,A -85,B 0,C 180,E1 10502.756,E2 10502.756} C_VEL
LIN {X 0,Y 409.614,Z 668.876,A -85,B 0,C 180,E1 10505.809,E2 10505.809} C_VEL
LIN {X 0,Y 405.026,Z 693.002,A -85,B 0,C 180,E1 10509.56,E2 10509.56} C_VEL
LIN {X 0,Y 401.164,Z 711.435,A -85,B 0,C 180,E1 10513.629,E2 10513.629} C_VEL
LIN {X 0,Y 398.295,Z 726.362,A -85,B 0,C 180,E1 10518.53,E2 10518.53} C_VEL
LIN {X 0,Y 396.836,Z 735.229,A -85,B 0,C 180,E1 10523.452,E2 10523.452} C_VEL
LIN {X 0,Y 396.376,Z 738.871,A -85,B 0,C 180,E1 10527.82,E2 10527.82} C_VEL
LIN {X 0,Y 396.384,Z 738.827,A -85,B 0,C 180,E1 10532.183,E2 10532.183} C_VEL
LIN {X 0,Y 396.925,Z 735.087,A -85,B 0,C 180,E1 10536.55,E2 10536.55} C_VEL
LIN {X 0,Y 398.353,Z 726.112,A -85,B 0,C 180,E1 10541.472,E2 10541.472} C_VEL
LIN {X 0,Y 401.095,Z 711.878,A -85,B 0,C 180,E1 10546.149,E2 10546.149} C_VEL
LIN {X 0,Y 405.088,Z 692.464,A -85,B 0,C 180,E1 10550.441,E2 10550.441} C_VEL
LIN {X 0,Y 409.718,Z 668.162,A -85,B 0,C 180,E1 10554.189,E2 10554.189} C_VEL
LIN {X 0,Y 413.825,Z 641.239,A -85,B 0,C 180,E1 10557.126,E2 10557.126} C_VEL
LIN {X 0,Y 405.633,Z 612.11,A -85,B 0,C 180,E1 10560.473,E2 10560.473} C_VEL
LIN {X 0,Y 393.173,Z 580.66,A -85,B 0,C 180,E1 10563.708,E2 10563.708} C_VEL
LIN {X 0,Y 393.035,Z 580.66,A -85,B 0,C 180,E1 10570.744,E2 10570.744} C_VEL
LIN {X 0,Y 393.04,Z 580.66,A -85,B 0,C 180,E1 10576.841,E2 10576.841} C_VEL
LIN {X 0,Y 393.05,Z 580.66,A -85,B 0,C 180,E1 10583.728,E2 10583.728} C_VEL
LIN {X 0,Y 393.166,Z 580.66,A -85,B 0,C 180,E1 10590.077,E2 10590.077} C_VEL
LIN {X 0,Y 393.425,Z 580.66,A -85,B 0,C 180,E1 10597.453,E2 10597.453} C_VEL
LIN {X 0,Y 393.617,Z 580.66,A -85,B 0,C 180,E1 10604.439,E2 10604.439} C_VEL
LIN {X 0,Y 393.938,Z 580.66,A -85,B 0,C 180,E1 10611.191,E2 10611.191} C_VEL
LIN {X 0,Y 394.461,Z 580.66,A -85,B 0,C 180,E1 10617.812,E2 10617.812} C_VEL
LIN {X 0,Y 394.229,Z 580.66,A -85,B 0,C 180,E1 10624.394,E2 10624.394} C_VEL
LIN {X 0,Y 393.945,Z 580.66,A -85,B 0,C 180,E1 10631.045,E2 10631.045} C_VEL
LIN {X 0,Y 393.634,Z 580.66,A -85,B 0,C 180,E1 10637.862,E2 10637.862} C_VEL
LIN {X 0,Y 393.352,Z 580.66,A -85,B 0,C 180,E1 10644.962,E2 10644.962} C_VEL
LIN {X 0,Y 393.136,Z 580.66,A -85,B 0,C 180,E1 10652.506,E2 10652.506} C_VEL
LIN {X 0,Y 393,Z 580.66,A -85,B 0,C 180,E1 10659.832,E2 10659.832} C_VEL
LIN {X 0,Y 393.06,Z 580.66,A -85,B 0,C 180,E1 10666.839,E2 10666.839} C_VEL
LIN {X 0,Y 393.098,Z 580.66,A -85,B 0,C 180,E1 10669.968,E2 10669.968} C_VEL
LIN {X 0,Y 414.832,Z 629.183,A -85,B 0,C 180,E1 10673.263,E2 10673.263} C_VEL
LIN {X 0,Y 418.938,Z 643.209,A -85,B 0,C 180,E1 10674.013,E2 10674.013} C_VEL
LIN {X 0,Y 415.467,Z 681.902,A -85,B 0,C 180,E1 10675.423,E2 10675.423} C_VEL
LIN {X 0,Y 410.997,Z 718.672,A -85,B 0,C 180,E1 10677.668,E2 10677.668} C_VEL
LIN {X 0,Y 406.312,Z 752.331,A -85,B 0,C 180,E1 10680.67,E2 10680.67} C_VEL
LIN {X 0,Y 401.859,Z 783.755,A -85,B 0,C 180,E1 10684.559,E2 10684.559} C_VEL
LIN {X 0,Y 398.478,Z 809.582,A -85,B 0,C 180,E1 10688.914,E2 10688.914} C_VEL
LIN {X 0,Y 396.418,Z 830.45,A -85,B 0,C 180,E1 10693.695,E2 10693.695} C_VEL
LIN {X 0,Y 395.544,Z 843.873,A -85,B 0,C 180,E1 10697.972,E2 10697.972} C_VEL
LIN {X 0,Y 392.92,Z 847.979,A -85,B 0,C 180,E1 10699.747,E2 10699.747} C_VEL
LIN {X 0,Y 387.505,Z 852.985,A -85,B 0,C 180,E1 10702.805,E2 10702.805} C_VEL
